// ---- Data types/Robot_udts/udt_GenericRobot_AnyFieldbus_OutputBytes_20220421.TcDUT
(*udt (user defined type) for all Fieldbus Based Robot Interfacing up to 64 Bytes
	Author(S): Brent Lekx-Toniolo of Sodecia GTAC;
	Version 1.0: November 2012
		- Initial Concept
	Version 20121204
		Changes from v1
			- Change to Naming Convention to include date as version
	Version 20220421
			- Changed starting point of Array fro 1 to 0 for TcHmi conventions, b.lekx-toniolo
*)
TYPE udt_GenericRobot_AnyFieldbus_OutputBytes_20220421 :
STRUCT
	Byte_: ARRAY [0..64] OF BYTE;
END_STRUCT
END_TYPE

// ---- Data types/Robot_udts/udt_GenericRobot_CycleTimes_20170304.TcDUT
(*udt (user defined type) for generic framework of cycle time counters for any robot
	Author(S): Brent Lekx-Toniolo of Sodecia GTAC;
	Version 20150622
		- Initila concept, BLT
	Version 20170304
		-added human, equip and total cycle time, JVD
*)
TYPE udt_GenericRobot_CycleTimes_20170304 :
STRUCT
	(*Cycle Times for Equipment Interf Zones*)
		Cycle_Time_OutEquip1: TIME;
		PrevCycle_Time_OutEquip1: TIME;
		Cycle_Time_OutEquip2: TIME;
		PrevCycle_Time_OutEquip2: TIME;
		Cycle_Time_OutEquip3: TIME;
		PrevCycle_Time_OutEquip3: TIME;
		Cycle_Time_OutEquip4: TIME;
		PrevCycle_Time_OutEquip4: TIME;
		Cycle_Time_OutEquip5: TIME;
		PrevCycle_Time_OutEquip5: TIME;
		Cycle_Time_OutEquip6: TIME;
		PrevCycle_Time_OutEquip6: TIME;
		Cycle_Time_OutEquip7: TIME;
		PrevCycle_Time_OutEquip7: TIME;
		Cycle_Time_OutEquip8: TIME;
		PrevCycle_Time_OutEquip8: TIME;

	(*Cycle Times for Human Interf Zones*)
		Cycle_Time_OutHuman1: TIME;
		PrevCycle_Time_OutHuman1: TIME;
		Cycle_Time_OutHuman2: TIME;
		PrevCycle_Time_OutHuman2: TIME;
		Cycle_Time_OutHuman3: TIME;
		PrevCycle_Time_OutHuman3: TIME;
		Cycle_Time_OutHuman4: TIME;
		PrevCycle_Time_OutHuman4: TIME;
		Cycle_Time_OutHuman5: TIME;
		PrevCycle_Time_OutHuman5: TIME;
		Cycle_Time_OutHuman6: TIME;
		PrevCycle_Time_OutHuman6: TIME;
		Cycle_Time_OutHuman7: TIME;
		PrevCycle_Time_OutHuman7: TIME;
		Cycle_Time_OutHuman8: TIME;
		PrevCycle_Time_OutHuman8: TIME;

		Cycle_Time_EquipTotal: TIME;
		Cycle_Time_HumanTotal: TIME;
		Cycle_Time_Total: TIME;

END_STRUCT
END_TYPE

// ---- Data types/Robot_udts/udt_Profibus_Motoman_Input.TcDUT
TYPE udt_Profibus_Motoman_Input :
	STRUCT
		Inputs:udt_ProfiNode_Status;
		(*Output Data From Robot*)
		SYS:UDINT;
		OG4: BYTE;
		OG5: BYTE;
		OG6: BYTE;
		OG7: BYTE;
		OG8: BYTE;
		OG9: BYTE;
		OG10: BYTE;
		OG11: BYTE;
		OG12: BYTE;
		OG13: BYTE;
		OG14: BYTE;
		OG15: BYTE;
		OG16: BYTE;
		OG17: BYTE;
		OG18: BYTE;
		OG19: BYTE;
		OG20: BYTE;
		OG21: BYTE;
		OG22: BYTE;
		OG23: BYTE;
		OG24: BYTE;
		OG25: BYTE;
		OG26: BYTE;
		OG27: BYTE;
		OG28: BYTE;
		OG29: BYTE;
		OG30: BYTE;
		OG31: BYTE;
		OG32: BYTE;
	END_STRUCT
END_TYPE

// ---- Data types/Robot_udts/udt_Profibus_Motoman_Input_20121204.TcDUT
(*udt (user defined type) for all Motoman Robot Controllers with HMS AnyBus Profibus Interface Card
	Author(S): Brent Lekx-Toniolo/Rob Remillard of Sodecia GTAC;
	Version 1.0: August 2010
		- Initial Concept
	Version 20121204
		Changes from v1
			- Increased Size to 32 Bytes
			- Change to Naming Convention to include date as version

	Last Edit: December 4th, 2012, blt
*)

TYPE udt_Profibus_Motoman_Input_20121204 :
	STRUCT
		Inputs:udt_ProfiNode_Status;
		(*Output Data From Robot, 32 Bytes total size*)
		SYS:UDINT;
		OG4: BYTE;
		OG5: BYTE;
		OG6: BYTE;
		OG7: BYTE;
		OG8: BYTE;
		OG9: BYTE;
		OG10: BYTE;
		OG11: BYTE;
		OG12: BYTE;
		OG13: BYTE;
		OG14: BYTE;
		OG15: BYTE;
		OG16: BYTE;
		OG17: BYTE;
		OG18: BYTE;
		OG19: BYTE;
		OG20: BYTE;
		OG21: BYTE;
		OG22: BYTE;
		OG23: BYTE;
		OG24: BYTE;
		OG25: BYTE;
		OG26: BYTE;
		OG27: BYTE;
		OG28: BYTE;
		OG29: BYTE;
		OG30: BYTE;
		OG31: BYTE;
		OG32: BYTE;
		OG33: BYTE;
	END_STRUCT
END_TYPE

// ---- Data types/Robot_udts/udt_Profibus_Motoman_Output.TcDUT
TYPE udt_Profibus_Motoman_Output :
	STRUCT
		(*Input Data To Robot*)
		SYS:UDINT;
		IG4:BYTE;
		IG5:BYTE;
		IG6:BYTE;
		IG7:BYTE;
		IG8:BYTE;
		IG9:BYTE;
		IG10:BYTE;
		IG11:BYTE;
		IG12:BYTE;
		IG13:BYTE;
		IG14:BYTE;
		IG15:BYTE;
		IG16:BYTE;
		IG17:BYTE;
		IG18:BYTE;
		IG19:BYTE;
		IG20:BYTE;
		IG21:BYTE;
		IG22:BYTE;
		IG23:BYTE;
		IG24:BYTE;
		IG25:BYTE;
		IG26:BYTE;
		IG27:BYTE;
		IG28:BYTE;
		IG29:BYTE;
		IG30:BYTE;
		IG31:BYTE;
		IG32:BYTE;
		END_STRUCT
END_TYPE

// ---- Data types/Robot_udts/udt_Profibus_Motoman_Output_20121204.TcDUT
(*udt (user defined type) for all Motoman Robot Controllers with HMS AnyBus Profibus Interface Card
	Author(S): Brent Lekx-Toniolo/Rob Remillard of Sodecia GTAC;
	Version 1.0: August 2010
		- Initial Concept
	Version 20121204
		Changes from v1
			- Increased Size to 32 Bytes
			- Change to Naming Convention to include date as version

	Last Edit: December 4th, 2012, blt
*)
TYPE udt_Profibus_Motoman_Output_20121204 :
	STRUCT
		(*Input Data To Robot, 32 Bytes total size*)
		SYS:UDINT;
		IG4:BYTE;
		IG5:BYTE;
		IG6:BYTE;
		IG7:BYTE;
		IG8:BYTE;
		IG9:BYTE;
		IG10:BYTE;
		IG11:BYTE;
		IG12:BYTE;
		IG13:BYTE;
		IG14:BYTE;
		IG15:BYTE;
		IG16:BYTE;
		IG17:BYTE;
		IG18:BYTE;
		IG19:BYTE;
		IG20:BYTE;
		IG21:BYTE;
		IG22:BYTE;
		IG23:BYTE;
		IG24:BYTE;
		IG25:BYTE;
		IG26:BYTE;
		IG27:BYTE;
		IG28:BYTE;
		IG29:BYTE;
		IG30:BYTE;
		IG31:BYTE;
		IG32:BYTE;
		IG33:BYTE;
		END_STRUCT
END_TYPE

// ---- Data types/Robot_udts/udt_SingleAxis_MoveData_20160908.TcDUT
(*udt (user defined type) to create data type for storing single Axis Movement Data Parameters:
	
	Author(S): Brent Lekx-Toniolo of Sodecia GTAC;

	Version 20150119
		- Initial Concept
	Version 20160908
		- Added Move_Type for vel vs pos type moves, b.lekx-toniolo


*)



TYPE udt_SingleAxis_MoveData_20160908 :
STRUCT
		Move_Type: UINT; 	(*Specify Move type during teaching*)
		Position: LREAL; 		(*Actual Stored Position Data*)
		Velocity: REAL; 		(*Target Velocity*)
		Accel: REAL; 			(*Target Acceleration Rate*)
		Decel: REAL;			(*Target Decceleration Rate*)
		End_Flag: BOOL;		(*Flag to Indicate Last Step In Program*)
END_STRUCT
END_TYPE

// ---- Data types/Robot_udts/udt_SingleAxis_Position_20150119.TcDUT
(*udt (user defined type) to create data type for storing single Axis Positional Data Parameters:
	
	Author(S): Brent Lekx-Toniolo of Sodecia GTAC;

	Version 20150119
		- Initial Concept

*)



TYPE udt_SingleAxis_Position_20150119 :
STRUCT
		Position: LREAL; 	(*Actual Stored Position Data*)
		Velocity: REAL; 	(*Target Velocity*)
		Accel: REAL; 		(*Target Acceleration Rate*)
		Decel: REAL;		(*Target Decceleration Rate*)
		End_Flag: BOOL;	(*Flag to Indicate Last Step In Program*)
END_STRUCT
END_TYPE

// ---- Data types/Schneider udts/udt_Schneider_VFD_20180808.TcDUT
(*udt (user defined type) for Schneider Electric VFD I/O Module
	Author(S): Justin Vandongen of Sodecia GTAC;

------------------------------------------------------------------------
	REVISION NOTES:

	Version 20180808
		- Initial Concept, j.vandongen
		- tested on ATV320 v1.11 ethercat module from schneider, j.vandongen

------------------------------------------------------------------------
*)

TYPE udt_Schneider_VFD_20180808 :
	STRUCT
	 	InfoData: udt_ECATSlave_Status;
	END_STRUCT
END_TYPE

// ---- Data types/Schneider udts/udt_Schneider_VFD_Image_20180808.TcDUT
(*udt (user defined type) for Schneider Electric VFD I/O Module
	Author(S): Justin Vandongen of Sodecia GTAC;

------------------------------------------------------------------------
	REVISION NOTES:

	Version 20180808
		- Initial Concept, j.vandongen
		- tested on ATV320 v1.11 ethercat module from schneider, j.vandongen
	Version 20250828
		- Added Cable breaks, r.jones
------------------------------------------------------------------------
*)

TYPE udt_Schneider_VFD_Image_20180808 :
	STRUCT
		
	VFD_State: udt_Schneider_VFD_20180808;
	Status_Word: UINT;
	Control_Word: UINT;
	Target_Velocity: INT;
	Move_TIME: TIME;
	ECAT_Cable_Breaks: UDINT;

	END_STRUCT
END_TYPE

// ---- Data types/Schneider udts/udt_Schneider_VFD_Inputs_20190123.TcDUT
(*udt (user defined type) for Schneider Electric VFD I/O Module
	Author(S): Justin Vandongen of Sodecia GTAC;

------------------------------------------------------------------------
	REVISION NOTES:

	Version 20180808
		- Initial Concept, j.vandongen
		- tested on ATV320 v1.11 ethercat module from schneider, j.vandongen
	Version 20190123
		- re-organized for more consistancy to generic device udts, b.lekx-toniolo

------------------------------------------------------------------------
*)

TYPE udt_Schneider_VFD_Inputs_20190123 :
	STRUCT
	InfoData: udt_ECATSlave_StatusEXT;

	Status_Word: UINT;
	Control_Effort: INT;
	Move_Time: TIME;

	END_STRUCT
END_TYPE

// ---- Data types/Schneider udts/udt_Schneider_VFD_Outputs_20190123.TcDUT
(*udt (user defined type) for Schneider Electric VFD I/O Module
	Author(S): Justin Vandongen of Sodecia GTAC;

------------------------------------------------------------------------
	REVISION NOTES:

	Version 20180808
		- Initial Concept, j.vandongen
		- tested on ATV320 v1.11 ethercat module from schneider, j.vandongen
	Version 20190123
		- re-organized for more consistancy to generic device udts, b.lekx-toniolo
------------------------------------------------------------------------
*)

TYPE udt_Schneider_VFD_Outputs_20190123 :
	STRUCT
	Control_Word: UINT;
	Target_Velocity: INT;
	END_STRUCT
END_TYPE

// ---- Data types/Servo Drive udts/AX5000 Diag/udt_AX5000Diag.TcDUT
(*Created by Beckhoff*)

TYPE udt_AX5000Diag :
STRUCT
	(* NC-Status *)
	nNCAxisID				: UDINT;
	bOperational				: BOOL;
	bC1DError				: BOOL;
	bWcStateError			: BOOL;
	bAxisError				: BOOL;
	iAxisErrorCode			: UDINT;

	(* Drive Diag *)
	strDriveType				: STRING(19);
	strMotorType				:STRING(31);
	wDriveStatus				: WORD;
	wClass1Diag				: WORD;
	stClass1Diag				: ST_AX5000_C1D;
	stDriveStatus				: ST_AX5000DriveStatus;
	stEcSlaveStateBits		: ST_EcSlaveStateBits;
	stEcSlaveState			: ST_EcSlaveState;
	bPreopToSafeOpError		: BOOL;
	bSafeOpToOpError		: BOOL;
	stCPxInvParamList			:ST_SoE_CPxInvParamList;
	iDiagNumber				: UDINT;
	stDiagNumberList			:ST_SoE_DiagNumList;
	strDiagMessage			: STRING(19);
	strDiagMessageFull		: STRING(60);
END_STRUCT
END_TYPE

// ---- Data types/Servo Drive udts/udt_AX5206_20160804.TcDUT
(*udt (user defined type) of Beckhoff AX5206 2 Axis Drive:
	auth. R.Remillard; 
	Oct 2014; version 1.0

	Version 20160804
		- Updated naming per convention, b.lekx-toniolo
		- Re-arranged variables for more consitent order with HW spec, b.lekx-toniolo
*)


TYPE udt_AX5206_20160804 :
STRUCT

	WcState:	BOOL;
	InfoData: udt_ECATSlave_StatusEXT;

END_STRUCT
END_TYPE

// ---- Data types/Servo Drive udts/udt_AX5805_20160804.TcDUT
(*udt (user defined type) of Beckhoff Type AX5805 Drive Safety Module:
	auth. R.Remillard; 
	October 2014; version 1.0

	Version 20160804
		- Updated naming per convention, b.lekx-toniolo
		- Re-arranged variables for more consitent order with HW spec, b.lekx-toniolo
	*)

TYPE udt_AX5805_20160804 :
STRUCT

	WcState:							BOOL;
 	InfoData: udt_ECATSlave_StatusEXT;

	FSOE_Command: 					USINT;
	Axis1_STO:						BOOL;
	Axis1_SSM1:						BOOL;
	Axis1_SSM2:						BOOL;
	Axis1_SOS1:						BOOL;
	Axis1_SSR1:						BOOL;
	Axis1_SDIp:						BOOL;
	Axis1_SDIn:						BOOL;
	Axis1_Error_Ack:					BOOL;
	FSOE_Slave_CRC_0:				UINT;
	Axis2_STO:						BOOL;
	Axis2_SSM1:						BOOL;
	Axis2_SSM2:						BOOL;
	Axis2_SOS1:						BOOL;
	Axis2_SSR1:						BOOL;
	Axis2_SDIp:						BOOL;
	Axis2_SDIn:						BOOL;
	Axis2_Error_Ack:					BOOL;
	FSOE_Slave_CRC_1:				UINT;
	FSOE_ConnID:					UINT;

	AMSAddress:						udt_AdsAddr_AX5805;

END_STRUCT
END_TYPE

// ---- Data types/Servo Drive udts/udt_AX5805_DiagData.TcDUT
TYPE udt_AX5805_DiagData :
STRUCT
	InternalDataA1:		UINT;	(*STO Reason Code Axis 1*)
	InternalDataA2:		UINT;	(*STO Reason Code Axis 2*)
	DiagDataA1:			UINT;	(*Ax5805 Setup Diagnositcs Axis 1*)
	DiagDataA2:			UINT;	(*AX5805 Setup Diagnostics Axis 2*)
	bError:				BOOL;
END_STRUCT
END_TYPE

// ---- Data types/Servo Drive udts/udt_EL7211_20150115.TcDUT
(*udt (user defined type) of Beckhoff - EL7211 series servo terminals:
	
	Author(S): Brent Lekx-Toniolo of Sodecia GTAC;

	Version 20150115
		- Initial Concept

*)


TYPE udt_EL7211_20150115 :
	STRUCT
		InfoData: udt_ECATSlave_Status;
	END_STRUCT
END_TYPE

// ---- Data types/SIC/udt_SIC_Profi_Input_20200727.TcDUT
TYPE udt_SIC_Profi_Input_20200727 :
STRUCT

			(*Status Of Profibus Slave*)
		Inputs:udt_ProfiNode_Status;
		(*Input Bytes*)
		Input0_0: ARRAY [0..15] OF USINT;
		Input0_1: ARRAY [0..15] OF USINT;
		Input0_2: ARRAY [0..15] OF USINT;
		Input0_3: ARRAY [0..15] OF USINT;
		Input0_4: ARRAY [0..15] OF USINT;
		Input0_5: ARRAY [0..15] OF USINT;
		Input0_6: ARRAY [0..15] OF USINT;
		Input0_7: ARRAY [0..15] OF USINT;
		Input0_8: ARRAY [0..15] OF USINT;
		Input0_9: ARRAY [0..15] OF USINT;
		Input0_10: ARRAY [0..15] OF USINT;
		Input0_11: ARRAY [0..15] OF USINT;
		Input0_12: ARRAY [0..15] OF USINT;
		Input0_13: ARRAY [0..15] OF USINT;
		Input0_14: ARRAY [0..15] OF USINT;
		Input0_15: ARRAY [0..15] OF USINT;

END_STRUCT
END_TYPE

// ---- Data types/SIC/udt_SIC_Profi_Output_20200727.TcDUT
TYPE udt_SIC_Profi_Output_20200727 :
STRUCT
	

		(*Input Bytes*)
		Output1_0: ARRAY [0..15] OF USINT;
		Output1_1: ARRAY [0..15] OF USINT;
		Output1_2: ARRAY [0..15] OF USINT;
		Output1_3: ARRAY [0..15] OF USINT;
		Output1_4: ARRAY [0..15] OF USINT;
		Output1_5: ARRAY [0..15] OF USINT;
		Output1_6: ARRAY [0..15] OF USINT;
		Output1_7: ARRAY [0..15] OF USINT;
		Output1_8: ARRAY [0..15] OF USINT;
		Output1_9: ARRAY [0..15] OF USINT;
		Output1_10: ARRAY [0..15] OF USINT;
		Output1_11: ARRAY [0..15] OF USINT;
		Output1_12: ARRAY [0..15] OF USINT;
		Output1_13: ARRAY [0..15] OF USINT;
		Output1_14: ARRAY [0..15] OF USINT;
		Output1_15: ARRAY [0..15] OF USINT;
		
END_STRUCT
END_TYPE

// ---- Data types/SmartRay/udt_PLC_Out_To_SmartRay_IN_20260119.TcDUT
(*udt of SmartRay profinet based
    PLC > Smart Ray 
  auth . Sodecia GTAC;
  Jan 2026: Version 1.0*)
TYPE udt_PLC_Out_To_SmartRay_IN_20260119 :
	
STRUCT
	(*Byte 0*)
	Byte_0 : BYTE;
	//PartType_In : BYTE;
	
	(*Byte 2-21*)
	Byte_2_21 : ARRAY[0..19] OF BYTE;
    //PartID_In : ARRAY[0..19] OF BYTE;
	
	(*Byte 24-43*)
	Byte_24_43 : ARRAY[0..19] OF BYTE;
	//PartIDVisu1_In : ARRAY[0..19] OF BYTE;
		
	(*Byte 44*)
	Byte_44 : BYTE;
	//Visu_NextPage_In : BOOL; (*Bit 4*)
	//Visu_NextWeld_In : BOOL; (*Bit 5*)
	//Visu_PreviousWeld_In : BOOL; (*Bit 6*)
	
	(*Byte 45*)
	Byte_45 : BYTE;
	//Visu_WorkerButton_In : BYTE; 
	
	(*Byte 48-67*)
	Byte_48_67 : ARRAY[0..19] OF BYTE;
	//PartIDVisu2_In : ARRAY[0..19] OF BYTE;
	
	(*Byte 68*)
	Byte_68 : BYTE;
	//Visu_NextPage2_In : BOOL; (*Bit 4*)
	//Visu_NextWeld2_In : BOOL; (*Bit 5*)
	//Visu_PreviousWeld2_In : BOOL; (*Bit 6*)

	(*Byte 69*)
	Byte_69 : BYTE;
	//Visu_WorkerButton2_In : BYTE;

END_STRUCT
END_TYPE

// ---- Data types/SmartRay/udt_Robot_Out_To_SmartRay_IN_20260119.TcDUT
TYPE udt_Robot_Out_To_SmartRay_IN_20260119 :
	// udt : Robot > Smart Ray
STRUCT
	(*Byte 0*)
	Reset_In : BOOL; (*Bit 0*)
	Alive_In : BOOL; (*Bit 1*)
	AutomaticMode_In : BOOL; (*Bit 2*)
 	SetupMode_In : BOOL; (*Bit 3*)
	
	(*Byte 1*)
	LaserOn_In : BOOL; (*Bit 1*)
	LaserOn2_In : BOOL; (*Bit 2*)
	SensortestOn_In : BOOL; (*Bit 3*)
	
	(*Byte 2*)
	InspectionCompleted_In : BOOL; (*Bit 2*)
	ToolfinderOn_In : BOOL; (*Bit 4*)

	(*Byte 3*)
	RobotSelection_In : BYTE;
	
	(*Byte 4-5*)
	JobID_In : UINT;
	
	(*Byte 6-7*)
	TrackSpeed_In : UINT;
	
END_STRUCT
END_TYPE

// ---- Data types/SmartRay/udt_SmartRay_Out_To_PLC_IN_20260119.TcDUT
(*udt of SmartRay profinet based
   Smart Ray > PLC 
  auth . Sodecia GTAC;
  Jan 2026: Version 1.0*)
TYPE udt_SmartRay_Out_To_PLC_IN_20260119 :
STRUCT
	(*Byte 0*)
	Byte_0 : BYTE;
	//PartType_Out : BYTE;
	
	(*Byte 2-21*)
	Byte_2_21 : ARRAY[0..19] OF BYTE;
	//PartID_Out : ARRAY[0..19] OF BYTE;
	
	(*Byte 22*)
	Byte_22 : BYTE;
	//QualityOK_Out_2 : BOOL; (*Bit 0*)
	//QualityNOK_Out_2 : BOOL; (*Bit 1*)
	//ResultValid_Out_2 : BOOL; (*Bit 2*)
	//LastTelegramSent_Out : BOOL; (*Bit 7*)
	
	(*Byte 24-43*)
	Byte_24_43 : ARRAY[0..19] OF BYTE;
	//PartIDVisu1_Out : ARRAY[0..19] OF BYTE;
	
	(*Byte 44*)
	Byte_44 : BYTE;
	(*WorkerResultOK_Out : BOOL; (*Bit 0*)
	WorkerResultNOK_Out : BOOL; (*Bit 1*)
	ReworkOK_Out : BOOL; (*Bit 2*)
	ReworkDone_Out : BOOL; (*Bit 3*)
	Visu_NextPage_Out : BOOL; (*Bit 4*)
	Visu_NextWeld_Out : BOOL; (*Bit 5*)
	Visu_PreviousWeld_Out : BOOL; (*Bit 6*)*)
	
	(*Byte 45*)
	Byte_45 : BYTE;
	//Visu_WorkerButon_Out :BYTE; 
	
	(*Byte 48-67*)
	Byte_48_67 : ARRAY[0..19] OF BYTE;
	//PartIDVisu2_Out : ARRAY[0..19] OF BYTE;
	
	(*Byte 68*)
	Byte_68 : BYTE;
	(*WorkerResultOK2_Out : BOOL; (*Bit 0*)
	WorkerResultNOK2_Out : BOOL; (*Bit 1*)
	ReworkOK2_Out : BOOL; (*Bit 2*)
	ReworkDone2_Out : BOOL; (*Bit 3*)
	Visu_NextPage2_Out : BOOL; (*Bit 4*)
	Visu_NextWeld2_Out : BOOL; (*Bit 5*)
	Visu_PreviousWeld2_Out : BOOL; (*Bit 6*)*)
	
	(*Byte 69*)
	Byte_69 : BYTE;
	//Vis_WorkerButton2_Out : BYTE;
	
	(*Byte 80-179*)
	Byte_80_179 : ARRAY[0..99] OF BYTE;
	//WeldResult_Out : ARRAY[0..99] OF BYTE;

END_STRUCT
END_TYPE

// ---- Data types/SmartRay/udt_SmartRay_Out_To_Robot_IN_20260119.TcDUT
(*udt of SmartRay profinet based
   Smart Ray > Robot 
  auth . Sodecia GTAC;
  Jan 2026: Version 1.0*)
TYPE udt_SmartRay_Out_To_Robot_IN_20260119 :	
STRUCT
	(*Status*)
	(*Byte 0*)
	SystemReady_Out : BOOL; (*Bit 0*)
	Alive_Out : BOOL; (*Bit 1*)
    FailureSystem_Out : BOOL; (*Bit 4*)
	FailureGlobal_Out : BOOL; (*Bit 5*)
	
	(*Byte 1*)
	SensorReady_Out : BOOL; (*Bit 0*)
	LaserOn_Out : BOOL; (*Bit 1*)
	LaserOn2_Out : BOOL; (*Bit 2*)
	SensortestOK_Out : BOOL; (*Bit 4*)
	SensortestNOK_Out : BOOL; (*Bit 5*)
	
	(*Byte 2*)
	QualityOK_Out : BOOL; (*Bit 0*)
	QualityNOK_Out : BOOL; (*Bit 1*)
	InspectionCompleted_Out : BOOL;(*Bit 2*)
	ResultValid_Out : BOOL; (*Bit 3*)
	ToolfinderValid_Out : BOOL; (*Bit 4*)
	ReferenceTrackSpeedActive_Out : BOOL; (*Bit 5*)
	
	(*Byte 3*)
	RobotSelection_Out : BYTE;
	
	(*Byte 4-5*)
	JobID_Out : UINT;
	
	(*Byte 6*)
	ErrorCode_Out : BYTE;
	
	(*Byte 7*)
	ToolfinderErrorCode_Out : BYTE;
	
	(*Byte 8-9*)
	Toolfinder_X : INT ;
	
	(*Byte 10-11*)
	Toolfinder_Y : INT;
	
	(*Byte 12-13*)
	Toolfinder_Z : INT;
	
	(*Byte 14-15*)
	Toolfinder_Q1_A_W :INT;
	
	(*Byte 16-17*)
	Toolfinder_Q2_B_P : INT;
	
	(*Byte 18-19*)
	Toolfinder_Q3_C_R : INT;
	
	(*Byte 20-21*)
	Toolfinder_Q4 : INT;
	
END_STRUCT
END_TYPE

// ---- Data types/SmartRay/UI udt/udt_SRxx_DiscreteImage.TcDUT
TYPE udt_SRxx_DiscreteImage :
STRUCT
	(*Smart Ray*)
	SR_Error : BOOL;
	SR_Comm_Error : BOOL;
	SR_PLC_FB_Error : BOOL;
	SR_Smart_Ray_OK : BOOL;
	SR_Smart_Ray_NOK : BOOL;
	
	Profinode_status : udt_ProfiNet_Status;

END_STRUCT
END_TYPE

// ---- Data types/SmartRay/UI udt/udt_SRxx_Input_Image.TcDUT
TYPE udt_SRxx_Input_Image :
STRUCT
	Retry : BOOL;
	Bypass :BOOL;
END_STRUCT
END_TYPE

// ---- Data types/SmartRay/UI udt/udt_SRxx_ToUI_20260122.TcDUT
TYPE udt_SRxx_ToUI_20260122 :
STRUCT
	DiscreteImage : udt_SRxx_DiscreteImage;
END_STRUCT
END_TYPE

// ---- Data types/SMC udts/udt_SMC_EX260_Stat.TcDUT
(*udt (user defined type) for SMC EX260 Serial Interface Valve Bank System EtherCAT Slave:
	auth. Brent Lekx-Toniolo of Toniolo Research & Development Inc.; 
	July 2010; version 1.0*)


TYPE udt_SMC_EX260_Stat :
STRUCT
	InfoData: udt_ECATSlave_Status;
END_STRUCT
END_TYPE

// ---- Data types/SMC udts/udt_SMC_EX260_ValveBank.TcDUT
(*udt (user defined type) for SMC EX260 Serial Interface Valve Bank System EtherCAT Slave:
	auth. Brent Lekx-Toniolo of Toniolo Research & Development Inc.; 
	August 2010; version 1.0*)


TYPE udt_SMC_EX260_ValveBank :
STRUCT
	Q: DINT;
END_STRUCT
END_TYPE

// ---- Data types/Trumpf udts/udt_EtherCat_Trumpf_InputWords_20171002.TcDUT

(*udt (user defined type) for all EtherCAT Based Trumpf Laser Interfacing on EL6692, up to 64 Bytes
	Author(S): Justin Vandongen of Sodecia GTAC;

------------------------------------------------------------------------
	REVISION NOTES:

	Version 20171002
		- Initial Concept, j.vandongen

------------------------------------------------------------------------
*)



TYPE udt_EtherCat_Trumpf_InputWords_20171002 :
STRUCT
	Laser_Out: ARRAY [0..9] OF WORD;
END_STRUCT
END_TYPE

// ---- Data types/Trumpf udts/udt_EtherCat_Trumpf_OutputWords_20171002.TcDUT

(*udt (user defined type) for all EtherCAT Based Trumpf Laser Interfacing on EL6692, up to 64 Bytes
	Author(S): Justin Vandongen of Sodecia GTAC;

------------------------------------------------------------------------
	REVISION NOTES:

	Version 20171002
		- Initial Concept, j.vandongen

------------------------------------------------------------------------
*)



TYPE udt_EtherCat_Trumpf_OutputWords_20171002 :
STRUCT
	Laser_In: ARRAY [0..9] OF WORD;
END_STRUCT
END_TYPE

// ---- Data types/Trumpf udts/udt_TrumpfImage_20171017.TcDUT

(*udt (user defined type) for all EtherCAT Based Trumpf Laser Discrete I/O Module
	Author(S): Justin Vandongen of Sodecia GTAC;

------------------------------------------------------------------------
	REVISION NOTES:

	Version 20171017
		- Initial Concept, j.vandongen

------------------------------------------------------------------------
*)


TYPE udt_TrumpfImage_20171017 :
STRUCT

		LSRT01: udt_EL6692_20121204;	(*EtherCAT bridge for Laser controller*)

		Program_REQ: UDINT;
		Program_ACK: UDINT;

		Light_Path_REQ: UDINT;
		Light_Path_ACK: UDINT;

		Laser_No_REQ: UDINT;
		Laser_No_ACK: UDINT;

		Laser_Power: UDINT;
		Laser_Power_Prev: UDINT;
		Energy: UDINT;
		Energy_Prev: UDINT;

		Weld_Complete: BOOL;
		Faulted: BOOL;


END_STRUCT
END_TYPE

// ---- Data types/UI udts/GTAC Component IO UI udts/udt_IVxx_ToUI_20250808.TcDUT
(*udt (user defined type) for interfacing to UI (User Interface)
this udt represents data that is passed from PLC to EACH UI

	Author(S): R.jones of Sodecia GTAC;
	- Initial Concept
	Version 20250723

*)

TYPE udt_IVxx_ToUI_20250808 :
	STRUCT

	(*Input and Output Data Images*)
	Discrete_Image: udt_IV2_DiscreteImage;
	(*EtherCAT Cable Break Flags*)
	ECAT_Cable_Breaks: UDINT;

	END_STRUCT
END_TYPE

// ---- Data types/UI udts/GTAC Component IO UI udts/udt_LSRxx_ToUI_20220224.TcDUT
(*udt (user defined type) for interfacing to UI (User Interface)
this udt represents data that is passed from PLC to EACH UI

	Author(S): Justin Vandongen of Sodecia GTAC;
	Version 20171011
		- Initial Concept
	Version 20220224
	- Overhaul during TcUI Migration project, b.lekx-toniolo / c.drees
*)

TYPE udt_LSRxx_ToUI_20220224:
	STRUCT

	(*Input and Output Data Images*)
	In_Image: udt_EtherCat_Trumpf_InputWords_20171002;
	Out_Image: udt_EtherCat_Trumpf_OutputWords_20171002;
	Discrete_Image: udt_TrumpfImage_20171017;

	(*EtherCAT Cable Break Flags*)
	ECAT_Cable_Breaks: UDINT;

	UI_FaultPrompts: UDINT;

	END_STRUCT
END_TYPE

// ---- Data types/UI udts/GTAC Component IO UI udts/udt_ESWxx_ToUI_20220224.TcDUT
(*udt (user defined type) for interfacing to UI (User Interface)
this udt represents data that is passed from PLC to EACH UI

	Author(S): Brent Lekx-Toniolo of Sodecia GTAC;
	Version 20150814
		- Initial Concept
	Version 20220224
	- Overhaul during TcUI Migration project, b.lekx-toniolo / c.drees

*)

TYPE udt_ESWxx_ToUI_20220224 :
	STRUCT

	(*Input and Output Data Images*)
	Discrete_Image: udt_ESWxx_Image_20150814;
	(*EtherCAT Cable Break Flags*)
	ECAT_Cable_Breaks: UDINT;

	END_STRUCT
END_TYPE

// ---- Data types/UI udts/GTAC Component IO UI udts/udt_ICxx_ToUI_20220224.TcDUT
(*udt (user defined type) for interfacing to UI (User Interface)
this udt represents data that is passed from PLC to EACH UI

	Author(S): Brent Lekx-Toniolo of Sodecia GTAC;
	Version 20141020
		- Initial Concept
	Version 20220224
	- Overhaul during TcUI Migration project, b.lekx-toniolo / c.drees

*)

TYPE udt_ICxx_ToUI_20220224 :
	STRUCT

	(*Input and Output Data Images*)
	Discrete_Image: udt_ICxx_Image;
	(*EtherCAT Cable Break Flags*)
	ECAT_Cable_Breaks: UDINT;

	END_STRUCT
END_TYPE

// ---- Data types/UI udts/GTAC Component IO UI udts/udt_MDxx_ToUI_20251008.TcDUT
(*udt (user defined type) for interfacing to UI (User Interface)
this udt represents data that is passed from PLC to EACH UI

	Author(S): Brent Lekx-Toniolo of Sodecia GTAC;
	Version 20150814
		- Initial Concept
	Version 20240926
	- Overhaul during TcUI Migration project, b.lekx-toniolo
	Version 20251008
	- MDxx instance update, b.lekx-toniolo
*)

TYPE udt_MDxx_ToUI_20251008 :
	STRUCT

	(*Input and Output Data Images*)
	Discrete_Image: udt_MDxx_Image_20251008;
	(*EtherCAT Cable Break Flags*)
	ECAT_Cable_Breaks: UDINT;

	END_STRUCT
END_TYPE

// ---- Data types/UI udts/GTAC Component IO UI udts/udt_NWxx_ToUI_20220224.TcDUT
(*udt (user defined type) for interfacing to UI (User Interface)
this udt represents data that is passed from PLC to EACH UI

	Author(S): Brent Lekx-Toniolo of Sodecia GTAC;
	Version 20141020
		- Initial Concept
	Version 20220224
	- Overhaul during TcUI Migration project, b.lekx-toniolo / c.drees

*)

TYPE udt_NWxx_ToUI_20220224 :
	STRUCT

	(*Input and Output Data Images*)
	Discrete_Image: udt_NWx_Image;
	(*EtherCAT Cable Break Flags*)
	ECAT_Cable_Breaks: UDINT;

	END_STRUCT
END_TYPE

// ---- Data types/UI udts/GTAC Component IO UI udts/udt_ISxx_ToUI_20241121.TcDUT
(*udt (user defined type) for interfacing to UI (User Interface)
this udt represents data that is passed from PLC to EACH UI

	Author(S): Brent Lekx-Toniolo of Sodecia GTAC;
	Version 20150813
		- Initial Concept
	Version 20220224
	- Overhaul during TcUI Migration project, b.lekx-toniolo / c.drees
	Version 20241121
		-PD to IS rename, as per GH SSCC610 repo Issue#162, b.lekx-toniolo

*)

TYPE udt_ISxx_ToUI_20241121 :
	STRUCT

	(*Input and Output Data Images*)
	Discrete_Image: udt_ISxx_Image_20241121;
	(*EtherCAT Cable Break Flags*)
	ECAT_Cable_Breaks: UDINT;
	END_STRUCT
END_TYPE

// ---- Data types/UI udts/GTAC Component IO UI udts/udt_ProdReportxx_ToUI_20220224.TcDUT
(*udt (user defined type) for interfacing to UI (User Interface)
this udt represents data that is passed from PLC to EACH UI

	Author(S): Brent Lekx-Toniolo of Sodecia GTAC;
	Version 20141021
		- Initial Concept
	Version 20160229
		- Updated udt instances, b.lekx-toniolo
	Version 20191125
		- Updated udt instances, b.lekx-toniolo
	Version 20220224
	- Overhaul during TcUI Migration project, b.lekx-toniolo / c.drees

*)

TYPE udt_ProdReportxx_ToUI_20220224 :
	STRUCT
	Curr_Prod_Report: udt_Generic_Production_20221007;
	Days_Prod_Report: udt_Generic_Production_20221007;
	Aft_Prod_Report: udt_Generic_Production_20221007;
	Mid_Prod_Report: udt_Generic_Production_20221007;

	END_STRUCT
END_TYPE

// ---- Data types/UI udts/GTAC Component IO UI udts/udt_Rxx_ToUI_20220224.TcDUT
(*udt (user defined type) for interfacing to UI (User Interface)
this udt represents data that is passed from PLC to EACH UI

	Author(S): Rob Remillard/Brent Lekx-Toniolo of Sodecia GTAC;
	Version 20121204
		- Initial Concept
		- For use with Generic Robot Image + ASSCV4.6, None SafeOP Discrete Image
	Version 20141020
		- Modified Name During Addition of more devices, b.lekx-toniolo
	Version 20150622
		- Added variables for passing of Interf Cycle Times, b.lekx-toniolo
	Version 20151028
		- Added discrete image type FSOE for V5.00 machine changes, b.lekx-toniolo
		- Added discrete image area for water stands, b.lekx-toniolo
	Version 20170531
		- Fronius Updates, b.lekx-toniolo
		- EOAT Instance Update, b.lekx-toniolo
	Version 20180418
		-EOAT instance removed, j.vandongen
	Version 20220224
	- Overhaul during TcUI Migration project, b.lekx-toniolo / c.drees

*)

TYPE udt_Rxx_ToUI_20220224 :
	STRUCT
	Robot_Type: UINT;
	(*General Data*)
	Status: UINT;
	Axis_Data: ARRAY [0..8] OF REAL;
 
	(*Input and Output Data Images*)
	In_Image: udt_GenericRobot_AnyFieldbus_InputBytes_20220421;
	Out_Image: udt_GenericRobot_AnyFieldbus_OutputBytes_20220421;
	Discrete_ImageFSOE: udt_RobotDiscreteNode_ImageFSOE_20151028;
	Discrete_ImageSSCCV46: udt_RobotDiscreteNode_ImageSSCCv46_20121204;
	Discrete_ImageSSCCV46wSAFEOP: udt_RobotDiscreteNode_ImageSSCCv46wSAFEOP_20131903;


	(*Option Configuration Inputs*)
	Options: udt_Generic_Robot_Options_20170531;
		(*Optional Equipment related to Robot*)
		WS_Discrete_Image: ARRAY [0..2] OF udt_WaterStand_Image_20220131;
		ATI_Discrete_Image: udt_ATIxx_Image_20151104;
		Reamer_Discrete_Image: udt_Reamerxx_Image_20180405;
		(*Robot Fronius Status Visualization*)
		Fronius_Status: udt_Fronius_Status_20170531;

	(*EtherCAT Cable Break Flags*)
	ECAT_Cable_Breaks: UDINT;
	(*Cycle Times*)
	CT: udt_GenericRobot_CycleTimes_20170304;
	(*Ped IO to be shown*)
	Ped_IO_ToShow: ARRAY [0..3] OF UINT;

	END_STRUCT
END_TYPE

// ---- Data types/UI udts/GTAC Component IO UI udts/udt_SDxx_ToUI_20220224.TcDUT
(*udt (user defined type) for interfacing to UI (User Interface)
this udt represents data that is passed from PLC to EACH UI

	Author(S): Rob Remillard/Brent Lekx-Toniolo of Sodecia GTAC;
	Version 2015 (Named udt_HMI_Input): August 2010
		- Initial Concept
	Version 20160804
		- Renamed to "...UI specific_SD...." for convention, b.lekx-toniolo
		- Added Data area for Positioning UI, b.lekx-toniolo
		- Updated instance of drive image as per it's naming update, b.lekx-toniolo
	Version 20220224
	- Overhaul during TcUI Migration project, b.lekx-toniolo / c.drees

*)

TYPE udt_SDxx_ToUI_20220224 :
	STRUCT

		(*Input and Output Data Images*)
		Discrete_Image:	udt_Drive_Image_20190816;
		(*EtherCAT Cable Break Flags*)
		ECAT_Cable_Breaks: UDINT;
		(*Confirm Axis Local Control Request*)
		AxisLocalControl_IC_ACKS: ARRAY[0..2] OF UINT;

	END_STRUCT
END_TYPE

// ---- Data types/UI udts/GTAC Component IO UI udts/udt_SLxx_ToUI_20220224.TcDUT
(*udt (user defined type) for interfacing to UI (User Interface)
this udt represents data that is passed from PLC to EACH UI

	Author(S): Brent Lekx-Toniolo of Sodecia GTAC;
	Version 20141020
		- Initial Concept
	Version 20220224
	- Overhaul during TcUI Migration project, b.lekx-toniolo / c.drees

*)

TYPE udt_SLxx_ToUI_20220224 :
	STRUCT

	(*Input and Output Data Images*)
	In_Image: udt_Graco_Input;
	Out_Image: udt_Graco_Outputs;
	(*Image for Profibus Master (Internal or External to Dispensing unit)*)
	Txx_ProfiMaster AT %I*: udt_EL6731;
	(*EtherCAT Cable Break Flags*)
	ECAT_Cable_Breaks: UDINT;


	END_STRUCT
END_TYPE

// ---- Data types/UI udts/GTAC Component IO UI udts/udt_SSxx_ToUI_20250704.TcDUT
(*udt (user defined type) for interfacing to UI (User Interface)
this udt represents data that is passed from PLC to EACH UI

	Author(S): Brent Lekx-Toniolo of Sodecia GTAC;
	Version 20150814
		- Initial Concept
	Version 20220224
	- Overhaul during TcUI Migration project, b.lekx-toniolo / c.drees

*)

TYPE udt_SSxx_ToUI_20250704 :
	STRUCT

	(*Input and Output Data Images*)
	Discrete_Image: udt_SSxx_Image_20250704;
	(*EtherCAT Cable Break Flags*)
	ECAT_Cable_Breaks: UDINT;

	END_STRUCT
END_TYPE

// ---- Data types/UI udts/GTAC Component IO UI udts/udt_STxx_ToUI_20220224.TcDUT
(*udt (user defined type) for interfacing to UI (User Interface)
this udt represents data that is passed from PLC to EACH UI

	Author(S): Brent Lekx-Toniolo of Sodecia GTAC;
	Version 20141020
		- Initial Concept
	Version 20200212
		- Updated Instances for Nelson to Emhart changes, b.lekx-toniolo
	Version 20220224
	- Overhaul during TcUI Migration project, b.lekx-toniolo / c.drees

*)

TYPE udt_STxx_ToUI_20220224 :
	STRUCT

	(*Input and Output Data Images*)
	In_Image: udt_Emhart_TE1500_Input;
	Out_Image: udt_Emhart_TE1500_Output;
	Discrete_Image: udt_STxx_DiscreteNode_20200212;
	(*EtherCAT Cable Break Flags*)
	ECAT_Cable_Breaks: UDINT;


	END_STRUCT
END_TYPE

// ---- Data types/UI udts/GTAC Component IO UI udts/udt_SDxx_FromUI_20220224.TcDUT
(*udt (user defined type) for interfacing to UI (User Interface)
this udt represents data that is passed from EACH UI to PLC

	Author(S): Brent Lekx-Toniolo of Sodecia GTAC;
	Version 20160811
		- Original Concept, b.lekx-toniolo
	Version 20220224
	- Overhaul during TcUI Migration project, b.lekx-toniolo / c.drees

*)
TYPE udt_SDxx_FromUI_20220224 :
STRUCT
		AxisLocalControl_IC_REQS: ARRAY[0..2] OF UINT;
		Mode_Select: ARRAY[0..2] OF INT;
		Error_Reset: ARRAY[0..2] OF BOOL;
		Program_Reset: ARRAY[0..2] OF BOOL;

		PlayBack_Speed_Percentage: ARRAY[0..2] OF REAL;
		Explicit_Step_REQ: ARRAY[0..2] OF UINT;
		Start_Explicit_StepCall: ARRAY[0..2] OF BOOL;
		Start_PlayBack: ARRAY[0..2] OF BOOL;
		Stop_PlayBack: ARRAY[0..2] OF BOOL;
		PlayBack_StepPermit: ARRAY[0..2] OF BOOL;


		Teach_Params: ARRAY[0..2] OF udt_SingleAxis_MoveData_20160908; (*Struct of Teach paramaeters*)
		Teach_Servo_HomePos: ARRAY[0..2] OF BOOL;
		Teach_JogFast_Plus: ARRAY[0..2] OF BOOL;
		Teach_JogFast_Minus: ARRAY[0..2] OF BOOL;
		Teach_JogSlow_Plus: ARRAY[0..2] OF BOOL;
		Teach_JogSlow_Minus: ARRAY[0..2] OF BOOL;
		Teach_Inch_Plus: ARRAY[0..2] OF BOOL;
		Teach_Inch_Minus: ARRAY[0..2] OF BOOL;
		Teach_MicroInch_Enable: ARRAY[0..2] OF BOOL;
		Teach_Record_CurrentPos: ARRAY[0..2] OF BOOL;
		Teach_ParamsOverwrite_Flag: ARRAY[0..2] OF BOOL;

END_STRUCT
END_TYPE

// ---- Data types/UI udts/GTAC Component IO UI udts/udt_VFDxx_ToUI_20250723.TcDUT
(*udt (user defined type) for interfacing to UI (User Interface)
this udt represents data that is passed from PLC to EACH UI

	Author(S): Rich Jones;
	Version 20250723
	- Initial Concept
	
*)

TYPE udt_VFDxx_ToUI_20250723 :
	STRUCT

	(*Input and Output Data Images*)
	Discrete_Image: udt_Schneider_VFD_Image_20180808;

	END_STRUCT
END_TYPE

// ---- Data types/UI udts/udt_UIcommon_InputPers_20250612.TcDUT
(*udt (user defined type) for interfacing to UI (User Interface)
this udt represents PERSISTENT data that is passed from ALL UIs to PLC

	Version 20191127
		- Cleaned up various, added structure and added production config variables, b.lekx-toniolo
	Version 20250612
		- Added in Nut Weld LVDT Config area to help reduce ground up work on nut weld applications, b.lekx-toniolo
*)

TYPE udt_UIcommon_InputPers_20250612 :
	STRUCT
(*Standard Persistent Inputs from UI*)
	(*Production Configuration*)
	ProdConfig_Common: udt_Generic_ShiftCommonConfig_20220420;
	ProdConfig_Day: udt_Generic_ShiftConfigUDINT_20160531;
	ProdConfig_Aft: udt_Generic_ShiftConfigUDINT_20160531;
	ProdConfig_Mid: udt_Generic_ShiftConfigUDINT_20160531;

(*Nut Weld based LVDT Configuration*)
	Config_NutWeld_LVDT: ARRAY [0..5] OF udt_Generic_NutWeldLVDTConfig_20250612;
	
(*General QA Configuration Items*)
	Config_Vision_Fail_Limits: ARRAY[0..16] OF  UINT;
	Config_NOK_BinCount_Limits: ARRAY[0..16] OF UINT;
	Config_NOK_Consecutive_Limits: ARRAY[0..16] OF UINT;
	
	
(*Add Non- Standard Persistent Inputs from UI here*)


	END_STRUCT
END_TYPE

// ---- Data types/UI udts/udt_UIcommon_Input_20250616.TcDUT
(*udt (user defined type) for interfacing to UI (User Interface)
this udt represents data that is passed from ALL UIs to PLC

	Author(S): Rob Remillard/Brent Lekx-Toniolo of Sodecia GTAC;
	Version 1.0 (Named udt_HMI_Input): August 2010
		- Initial Concept
	Version 20141014
		- Increase for 30 Robot framework + Fix Renaming, b.lekx-toniolo
	Version 20150519
		- Added Report_Trigger_Reqs, b.lekx-toniolo
		- Added Rxx_ToolChange_Reqs, b.lekx-toniolo
	Version 20161129
		-Custom Setup for SIC marking, RRemillard
	Version 20161206
		-added Sealer bits, J.vandongen
	Version 20170626
		- added local dry cycle enables, b.lekx-toniolo / c.drees (edge automation)
	Version 20170801
		-added bit to control monitoring spaces from plc, RRemillard
	Version 20170804
		-added cycle hold, j.vandongen
	Version 20200611
		- added Rxx_Dress_Req, j.vandongen
	Version 20220224
		- overhaul during TcUI migration project, b.lekx-toniolo / c.drees
	Version 20240620
		- added rxx_tracctcp_req,  w. griffiths / b.lekx-toniolo 
	Version 20250616
		- Added in Nut Weld Based LVDT Input Image, b.lekx-toniolo	

*)

TYPE udt_UIcommon_Input_20250616 :
	STRUCT
(*Standard Inputs from UI*)
	(*Common to Cell*)
	StartRobots: BOOL;
	StopRobots: BOOL;
	Cycle_Hold: BOOL;
	RelaseSGK1: BOOL;
	RelaseSGK2: BOOL;
	LockSGK1: BOOL;
	LockSGK2: BOOL;
	ControlPower1: BOOL;
	ControlPower2: BOOL;
	Force_TipChange: BOOL;
	TipChange_Complete: BOOL;
	Reset_ChangeCount: BOOL;
	Enable_Dry_Cycle: BOOL;
	Local_DryCycle_Enables: UDINT;
	QA_Request_LH: BOOL;
	QA_Request_RH: BOOL;
	QA_Reinsert_LH: BOOL;
	QA_Reinsert_RH: BOOL;
	QA_Reset: UINT;
	QA_NOK_BinCount_Resets: UINT;	
	QA_NOK_Consecutive_Resets: UINT;
	
	Global_Robot_Speed: BYTE;
	Low_Speed_Req: BOOL;
	Force_Master_Test: BOOL;
	Force_Brake_Test: BOOL;
	Bypass_REQS: UDINT;
	CustomApplication_REQS: UDINT;
	Rxx_ToolChange_REQS: UDINT;
	T1_Zone_Test: BOOL;
	Production_Report_Trigger_ACKS: UDINT;
	Product_Report_Trigger_ACKS: UDINT;

	(*Sealer Related Bits*)
	SL01_Purge_REQS: UINT;
	SL02_Purge_REQS: UINT;
	SL03_Purge_REQS: UINT;
	SL04_Purge_REQS: UINT;
	SL01_Dispense_Bypass: UINT;
	SL02_Dispense_Bypass: UINT;
	SL03_Dispense_Bypass: UINT;
	SL04_Dispense_Bypass: UINT;



(*Standard UI Control For Operator Stations and Status of TWCAT Driver Sheet Comms*)
	(*IC01*)
	IC01_Requests: INT;				(*Bit 1 = Production, 2 = Materials, 3 = Maintenance*)
	IC01_COMM_STAT: INT;			(*Communication Status of Twincat driver sheet in Indusoft*)
	(*IC02*)
	IC02_Requests: INT;				(*Bit 1 = Production, 2 = Materials, 3 = Maintenance*)
	IC02_COMM_STAT: INT;			(*Communication Status of Twincat driver sheet in Indusoft*)
	(*IC03*)
	IC03_Requests: INT;				(*Bit 1 = Production, 2 = Materials, 3 = Maintenance*)
	IC03_COMM_STAT: INT;			(*Communication Status of Twincat driver sheet in Indusoft*)
	(*IC04*)
	IC04_Requests: INT;				(*Bit 1 = Production, 2 = Materials, 3 = Maintenance*)
	IC04_COMM_STAT: INT;			(*Communication Status of Twincat driver sheet in Indusoft*)
	(*IC05*)
	IC05_Requests: INT;				(*Bit 1 = Production, 2 = Materials, 3 = Maintenance*)
	IC05_COMM_STAT: INT;			(*Communication Status of Twincat driver sheet in Indusoft*)
	(*IC06*)
	IC06_Requests: INT;				(*Bit 1 = Production, 2 = Materials, 3 = Maintenance*)
	IC06_COMM_STAT: INT;			(*Communication Status of Twincat driver sheet in Indusoft*)
	(*IC07*)
	IC07_Requests: INT;				(*Bit 1 = Production, 2 = Materials, 3 = Maintenance*)
	IC07_COMM_STAT: INT;			(*Communication Status of Twincat driver sheet in Indusoft*)
	(*IC08*)
	IC08_Requests: INT;				(*Bit 1 = Production, 2 = Materials, 3 = Maintenance*)
	IC08_COMM_STAT: INT;			(*Communication Status of Twincat driver sheet in Indusoft*)

(*Specific Inputs from UI*)
	(*Robot Control*)
	Rxx_Weld_Inhibit: BOOL;
	Rxx_Dress_Req: BOOL;
	Rxx_TraccTCP_Req: BOOL;
	R1_Weld_Inhibit: BOOL;
	R1_Disable_Power: BOOL;
	R1_Temp_Start: BOOL;
	R1_Dress_Req: BOOL;
	R1_TraccTCP_Req: BOOL;
	R2_Weld_Inhibit: BOOL;
	R2_Disable_Power: BOOL;
	R2_Temp_Start: BOOL;
	R2_Dress_Req: BOOL;
	R2_TraccTCP_Req: BOOL;
	R3_Weld_Inhibit: BOOL;
	R3_Disable_Power: BOOL;
	R3_Temp_Start: BOOL;
	R3_Dress_Req: BOOL;
	R3_TraccTCP_Req: BOOL;
	R4_Weld_Inhibit: BOOL;
	R4_Disable_Power: BOOL;
	R4_Temp_Start: BOOL;
	R4_Dress_Req: BOOL;
	R4_TraccTCP_Req: BOOL;
	R5_Weld_Inhibit: BOOL;
	R5_Disable_Power: BOOL;
	R5_Temp_Start: BOOL;
	R5_Dress_Req: BOOL;
	R5_TraccTCP_Req: BOOL;
	R6_Weld_Inhibit: BOOL;
	R6_Disable_Power: BOOL;
	R6_Temp_Start: BOOL;
	R6_Dress_Req: BOOL;
	R6_TraccTCP_Req: BOOL;
	R7_Weld_Inhibit: BOOL;
	R7_Disable_Power: BOOL;
	R7_Temp_Start: BOOL;
	R7_Dress_Req: BOOL;
	R7_TraccTCP_Req: BOOL;
	R8_Weld_Inhibit: BOOL;
	R8_Disable_Power: BOOL;
	R8_Temp_Start: BOOL;
	R8_Dress_Req: BOOL;
	R8_TraccTCP_Req: BOOL;
	R9_Weld_Inhibit: BOOL;
	R9_Disable_Power: BOOL;
	R9_Temp_Start: BOOL;
	R9_Dress_Req: BOOL;
	R9_TraccTCP_Req: BOOL;
	R10_Weld_Inhibit: BOOL;
	R10_Disable_Power: BOOL;
	R10_Temp_Start: BOOL;
	R10_Dress_Req: BOOL;
	R10_TraccTCP_Req: BOOL;
	R11_Weld_Inhibit: BOOL;
	R11_Disable_Power: BOOL;
	R11_Temp_Start: BOOL;
	R11_Dress_Req: BOOL;
	R11_TraccTCP_Req: BOOL;
	R12_Weld_Inhibit: BOOL;
	R12_Disable_Power: BOOL;
	R12_Temp_Start: BOOL;
	R12_Dress_Req: BOOL;
	R12_TraccTCP_Req: BOOL;
	R13_Weld_Inhibit: BOOL;
	R13_Disable_Power: BOOL;
	R13_Temp_Start: BOOL;
	R13_Dress_Req: BOOL;
	R13_TraccTCP_Req: BOOL;
	R14_Weld_Inhibit: BOOL;
	R14_Disable_Power: BOOL;
	R14_Temp_Start: BOOL;
	R14_Dress_Req: BOOL;
	R14_TraccTCP_Req: BOOL;
	R15_Weld_Inhibit: BOOL;
	R15_Disable_Power: BOOL;
	R15_Temp_Start: BOOL;
	R15_Dress_Req: BOOL;
	R15_TraccTCP_Req: BOOL;
	R16_Weld_Inhibit: BOOL;
	R16_Disable_Power: BOOL;
	R16_Temp_Start: BOOL;
	R16_Dress_Req: BOOL;
	R16_TraccTCP_Req: BOOL;
	R17_Weld_Inhibit: BOOL;
	R17_Disable_Power: BOOL;
	R17_Temp_Start: BOOL;
	R17_Dress_Req: BOOL;
	R17_TraccTCP_Req: BOOL;
	R18_Weld_Inhibit: BOOL;
	R18_Disable_Power: BOOL;
	R18_Temp_Start: BOOL;
	R18_Dress_Req: BOOL;
	R18_TraccTCP_Req: BOOL;
	R19_Weld_Inhibit: BOOL;
	R19_Disable_Power: BOOL;
	R19_Temp_Start: BOOL;
	R19_Dress_Req: BOOL;
	R19_TraccTCP_Req: BOOL;
	R20_Weld_Inhibit: BOOL;
	R20_Disable_Power: BOOL;
	R20_Temp_Start: BOOL;
	R20_Dress_Req: BOOL;
	R20_TraccTCP_Req: BOOL;
	R21_Weld_Inhibit: BOOL;
	R21_Disable_Power: BOOL;
	R21_Temp_Start: BOOL;
	R21_Dress_Req: BOOL;
	R21_TraccTCP_Req: BOOL;
	R22_Weld_Inhibit: BOOL;
	R22_Disable_Power: BOOL;
	R22_Temp_Start: BOOL;
	R22_Dress_Req: BOOL;
	R22_TraccTCP_Req: BOOL;
	R23_Weld_Inhibit: BOOL;
	R23_Disable_Power: BOOL;
	R23_Temp_Start: BOOL;
	R23_Dress_Req: BOOL;
	R23_TraccTCP_Req: BOOL;
	R24_Weld_Inhibit: BOOL;
	R24_Disable_Power: BOOL;
	R24_Temp_Start: BOOL;
	R24_Dress_Req: BOOL;
	R24_TraccTCP_Req: BOOL;
	R25_Weld_Inhibit: BOOL;
	R25_Disable_Power: BOOL;
	R25_Temp_Start: BOOL;
	R25_Dress_Req: BOOL;
	R25_TraccTCP_Req: BOOL;
	R26_Weld_Inhibit: BOOL;
	R26_Disable_Power: BOOL;
	R26_Temp_Start: BOOL;
	R26_Dress_Req: BOOL;
	R26_TraccTCP_Req: BOOL;
	R27_Weld_Inhibit: BOOL;
	R27_Disable_Power: BOOL;
	R27_Temp_Start: BOOL;
	R27_Dress_Req: BOOL;
	R27_TraccTCP_Req: BOOL;
	R28_Weld_Inhibit: BOOL;
	R28_Disable_Power: BOOL;
	R28_Temp_Start: BOOL;
	R28_Dress_Req: BOOL;
	R28_TraccTCP_Req: BOOL;
	R29_Weld_Inhibit: BOOL;
	R29_Disable_Power: BOOL;
	R29_Temp_Start: BOOL;
	R29_Dress_Req: BOOL;
	R29_TraccTCP_Req: BOOL;
	R30_Weld_Inhibit: BOOL;
	R30_Disable_Power: BOOL;
	R30_Temp_Start: BOOL;
	R30_Dress_Req: BOOL;
	R30_TraccTCP_Req: BOOL;

	(*Fixture Control*)
	Fix01_Discrete_In: udt_FixXX_Input_Image_20180202;
	Fix02_Discrete_In: udt_FixXX_Input_Image_20180202;
	Fix03_Discrete_In: udt_FixXX_Input_Image_20180202;
	Fix04_Discrete_In: udt_FixXX_Input_Image_20180202;
	Fix05_Discrete_In: udt_FixXX_Input_Image_20180202;
	Fix06_Discrete_In: udt_FixXX_Input_Image_20180202;
	Fix07_Discrete_In: udt_FixXX_Input_Image_20180202;
	Fix08_Discrete_In: udt_FixXX_Input_Image_20180202;
	Fix09_Discrete_In: udt_FixXX_Input_Image_20180202;
	Fix10_Discrete_In: udt_FixXX_Input_Image_20180202;
	Fix11_Discrete_In: udt_FixXX_Input_Image_20180202;
	Fix12_Discrete_In: udt_FixXX_Input_Image_20180202;
	Fix13_Discrete_In: udt_FixXX_Input_Image_20180202;
	Fix14_Discrete_In: udt_FixXX_Input_Image_20180202;
	Fix15_Discrete_In: udt_FixXX_Input_Image_20180202;
	Fix16_Discrete_In: udt_FixXX_Input_Image_20180202;

	Fix101_Discrete_In: udt_FixXX_Input_Image_20180202;
	Fix102_Discrete_In: udt_FixXX_Input_Image_20180202;
	Fix103_Discrete_In: udt_FixXX_Input_Image_20180202;
	Fix104_Discrete_In: udt_FixXX_Input_Image_20180202;
	Fix105_Discrete_In: udt_FixXX_Input_Image_20180202;
	Fix106_Discrete_In: udt_FixXX_Input_Image_20180202;
	Fix107_Discrete_In: udt_FixXX_Input_Image_20180202;
	Fix108_Discrete_In: udt_FixXX_Input_Image_20180202;
	Fix109_Discrete_In: udt_FixXX_Input_Image_20180202;
	Fix110_Discrete_In: udt_FixXX_Input_Image_20180202;
	Fix111_Discrete_In: udt_FixXX_Input_Image_20180202;
	Fix112_Discrete_In: udt_FixXX_Input_Image_20180202;

	(*Nut Weld based LVDTs*)
	NutWeld_LVDT_Discrete_In: ARRAY [0..5] OF udt_NutWeldLVDT_Input_Image_20250616;
	
	(*Custom addition for SIC marking units*)
	SIC01_BypassReq: BOOL;
	SIC02_BypassReq: BOOL;


	(*Generic Servo Control*)
	SD: ARRAY [0..30] OF udt_SDxx_FromUI_20220224;
	
	(*IV2/3 UI Inputs*)
	IVx_Discrete_In: ARRAY [0..5] OF udt_IVxx_Input_Image_20250812;
	
	(*SRxx*)
	SRx_Discrete_In : ARRAY [0..1] OF udt_SRxx_Input_Image;	

	END_STRUCT
END_TYPE

// ---- Data types/UI udts/udt_UIcommon_Output_20251008.TcDUT
(*udt (user defined type) for interfacing to UI (User Interface)
this udt represents data that is passed from PLC to ALL UIs

	Author(S): Rob Remillard/Brent Lekx-Toniolo of Sodecia GTAC;
	Version 1.0 (Named udt_HMI_Output): August 2010
		- Initial Concept
	Version 20141014
		- Increase for 30 Robot framework + Fix Renaming, b.lekx-toniolo
	Version 20141128
		- Added ESW Count Option, b.lekx-toniolo
		- Added More WSxxs, b.lekx-toniolo
	Version 20141209
		- Added TTxx Ints for location indexes of Turntables, b.lekx-toniolo
	Version 20141211
		- Added SMB Image, b.lekx-toniolo
		- Updated Ecat Master Instance, b.lekx-toniolo
	Version 20150226
		- Added Target Cycle Time for display on UI screen(s), b.lekx-toniolo
	Version 20150812
		- Added PD Count for display on UI screen(s), b.lekx-toniolo
	Version 20150827
		- Renamed Option_HumanFix_Count to Option_HumanFix_Enables, b.lekx-toniolo
	Version 20160113
		- Increased fault area size and added area for water setpoint options, b.lekx-toniolo
		- Added UI Prompt flags for controls faults prompting , b.lekx-toniolo
	Version 20160418
		- Added Area for Robot Water Flow Timeout feature configuration data, b.lekx-toniolo
		- updated ECAT Master area to include new new image with HW config data, b.lekx-toniolo 
	Version 20160519
		-Added udts for Each Shift Structure Configuration, b.lekx-toniolo
		- Removed Old Model Change Allow Bools, b.lekx-toniolo
		- Added Report_Trigger_Acks, b.lekx-toniolo
		- Added Rxx_ToolChange_Acks, b.lekx-toniolo
	Version 20161129
		-Custom setup for SIC marking, RRemillard	
	Version 20161206
		-added sealer bits, j.vandongen
	Version 20170626
		- added local dry cycle, b.lekx-toniolo / c.drees (edge automation)
	Version 20170801
		-added bit to control monitoring spaces from plc, RRemillard
	Version 20170804
		-added cycle hold ack, j.vandongen
	Version 20180417	
		-added Option_EOAT_Count, j.vandongen
		-added Option_LaserController, j.vandongen
		-changed var type Config_Fault, j.vandongen
		-added EOAT discrete images, j.vandongen
		-added SD option count, j.vandongen
	Version 20191125
		- Added ProdConfig_Common, b.lekx-toniolo 
		- Update names for EOAT -> UI interface to correct naming mismatch in UI driver sheet, b.lekx-toniolo
	Version 20191210
		-Added Code to deal with TC3 Changes:
			-Motherboard data is no longer a device in the I/O tree and MUST be read in from the MDP.  Not all data is available anymore, so UDT modified
				to show data changes
			-Application data is no longer stored in the same global system variable as before, new structure added for the App data
			-Task Data is no longer stored in the same global system variable as before, new strucuture added for the task data.
	Version 20220224
		- Overhaul during TcUI migration project, b.lekx-toniolo / c.drees
		- Added in In_Sim_Mode for integration into simulation, b.lekx-toniolo	
	Version 20240909
		- Increased Product Report Data Area to give EOATs a storage location, b.lekx-toniolo	
	Version 20240926
		- Added in data area for MDxx (Motorized Door) component, b.lekx-toniolo	
	Version 20241121
		- PD to IS rename, as per GH SSCC610 repo Issue#162, b.lekx-toniolo
	Version 20250616
		- Added in Nut Weld Based LVDT Output Image, b.lekx-toniolo	
	Version 20250716
		- Added in Exceed_Counter_Value, per SSCC610 GH Issue #235, b.lekx-toniolo
	Version 20250723
		- Added in config count and general discrete images for VFD additions, b.lekx-toniolo / r. jones
	Version20251008
		- MDxx instance update, b.lekx-toniolo	
*)

TYPE udt_UIcommon_Output_20251008 :
	STRUCT
(*Configuration Data to UI*)
	Machine_Serial: STRING;
	Machine_Common_Name: STRING;
	Machine_Build_Used: STRING;
	Machine_Appl_Dev: STRING;
	
	ProdConfig_Target_CycleTime: TIME;

	ProdConfig_Common: udt_Generic_ShiftCommonConfig_20220420;
	ProdConfig_Day: udt_Generic_ShiftConfigUDINT_20160531;
	ProdConfig_Aft: udt_Generic_ShiftConfigUDINT_20160531;
	ProdConfig_Mid: udt_Generic_ShiftConfigUDINT_20160531;

	Option_Air1: BOOL;
	Option_Air2: BOOL;
	Option_Water1: BOOL;
	Option_Water2: BOOL;

	Option_WaterTimeOut_Enable: BOOL;
	Option_WaterFlowTimeOut_SP: TIME;
	Option_WaterTempHighLimit1: REAL;
	Option_WaterFlowLowLimit1: REAL;
	Option_WaterTempHighLimit2: REAL;
	Option_WaterFlowLowLimit2: REAL;

	Option_IS_Count: UINT;
	Option_ESW_Count: UINT;
	Option_MD_Count: UINT;
	Option_IC_Count: UINT;
	Option_HumanFix_Enables: UDINT;
	Option_InternalFix_Count: UINT;
	Option_Robot_Count: UINT;
	Option_Ped_Count: UINT;
	Option_StudController_Count: UINT;
	Option_SealController_Count: UINT;
	Option_NutWelder_Count: UINT;
	Option_EOAT_Count: UINT;
	Option_LaserController_Count: UINT;
	Option_SD_Count: UINT;
	Option_VFD_Count: UINT;
	Config_Fault:UDINT;

(*Standard Outputs to UI*)
	(*Common to Cell*)
	ControlPower1_OK: BOOL; (*Control Power is ON*)
	ControlPower2_OK: BOOL;	(*spare*)
	CycleHold_OK: BOOL;
	Estops_OK: BOOL;		(*All Estops OK and Reset*)
	Safety_Gates_OK: BOOL;	(*All Safety Gates OK and Reset*)
	Faults_OK: BOOL;		(*No Major Faults*)
	TipChangeReq_OK: BOOL;
	TipChangeComp_OK: BOOL;
	Change_Count: INT;
	TipChange_Part_Count: INT;
	InDryCycle:BOOL;
	In_Local_DryCycle:UDINT;
	Allow_Model_Change: BOOL;
	QA_LH_Ready: BOOL;
	QA_RH_Ready: BOOL;
	QA_NOK_BinCounts: ARRAY [0..16] OF UINT;
	Spare1: BOOL;
	Spare2: BOOL;
	SMB_Status_Image: udt_SMB_Status_20141211;
	EtherCat_Master_Image: udt_ECATMaster_Image_20220224;
	EL6900_FB_Errors1: DINT;
	EL6900_Comm_Errors1: DINT;
	EL6900_Out_Errors1: DINT;
	EL6900_FB_Errors2: DINT;
	EL6900_Comm_Errors2: DINT;
	EL6900_Out_Errors2: DINT;
	Overall_Controls_Fault: UINT;
	In_Low_Speed: BOOL;
	Under_Construction: BOOL;	(*System is Under Construction*)
	In_Sim_Mode: BOOL; 			(*System in Simulation mode, added during project 90034*)
	MasterTest_Req_OK: BOOL;
	BrakeTest_Req_OK: BOOL;
	Rxx_ReadyFor_TipChange: UDINT;
	Bypass_ACKS: UDINT;
	CustomApplication_ACKS: UDINT;
	Rxx_ToolChange_ACKS: UDINT;
	T1_Zone_Test_ACK: BOOL;
	Production_Report_Trigger_REQS: UDINT;
	Product_Report_Trigger_REQS: UDINT;

	(* TC3 Specific data types for App data, Task data and Motherboard Diagnostics *)
	Appdata 	:PlcAppSystemInfo;
	TaskData	:PlcTaskSystemInfo;
	MboardData	:udt_HardwareDiags;
	Exceed_Counter_Value: UDINT;
	
	(*Sealer Bits*)
	SL01_Dispense_Count: UINT;
	SL02_Dispense_Count: UINT;
	SL03_Dispense_Count: UINT;
	SL04_Dispense_Count: UINT;
	SL01_Bypass_ACK: UINT;
	SL02_Bypass_ACK: UINT;
	SL03_Bypass_ACK: UINT;
	SL04_Bypass_ACK: UINT;


(*Standard UI Visualization For Operator Stations*)
	(*IC01*)
	IC01OP1_LCHVR: BOOL;
	IC01OP1_LCHHR: BOOL;
	IC01OP1_LCRVR: BOOL;
	IC01OP2_LCHVR: BOOL;
	IC01OP2_LCHHR: BOOL;
	IC01OP2_LCRVR: BOOL;
	(*IC02*)
	IC02OP1_LCHVR: BOOL;
	IC02OP1_LCHHR: BOOL;
	IC02OP1_LCRVR: BOOL;
	IC02OP2_LCHVR: BOOL;
	IC02OP2_LCHHR: BOOL;
	IC02OP2_LCRVR: BOOL;
	(*IC03*)
	IC03OP1_LCHVR: BOOL;
	IC03OP1_LCHHR: BOOL;
	IC03OP1_LCRVR: BOOL;
	IC03OP2_LCHVR: BOOL;
	IC03OP2_LCHHR: BOOL;
	IC03OP2_LCRVR: BOOL;
	(*IC04*)
	IC04OP1_LCHVR: BOOL;
	IC04OP1_LCHHR: BOOL;
	IC04OP1_LCRVR: BOOL;
	IC04OP2_LCHVR: BOOL;
	IC04OP2_LCHHR: BOOL;
	IC04OP2_LCRVR: BOOL;
	(*IC05*)
	IC05OP1_LCHVR: BOOL;
	IC05OP1_LCHHR: BOOL;
	IC05OP1_LCRVR: BOOL;
	IC05OP2_LCHVR: BOOL;
	IC05OP2_LCHHR: BOOL;
	IC05OP2_LCRVR: BOOL;
	(*IC06*)
	IC06OP1_LCHVR: BOOL;
	IC06OP1_LCHHR: BOOL;
	IC06OP1_LCRVR: BOOL;
	IC06OP2_LCHVR: BOOL;
	IC06OP2_LCHHR: BOOL;
	IC06OP2_LCRVR: BOOL;
	(*IC07*)
	IC07OP1_LCHVR: BOOL;
	IC07OP1_LCHHR: BOOL;
	IC07OP1_LCRVR: BOOL;
	IC07OP2_LCHVR: BOOL;
	IC07OP2_LCHHR: BOOL;
	IC07OP2_LCRVR: BOOL;
	(*IC08*)
	IC08OP1_LCHVR: BOOL;
	IC08OP1_LCHHR: BOOL;
	IC08OP1_LCRVR: BOOL;
	IC08OP2_LCHVR: BOOL;
	IC08OP2_LCHHR: BOOL;
	IC08OP2_LCRVR: BOOL;


	(*Location Index for Animation of Turntables*)
	TT01_Location_Index: INT;
	TT02_Location_Index: INT;
	TT03_Location_Index: INT;
	TT04_Location_Index: INT;
	TT05_Location_Index: INT;
	TT06_Location_Index: INT;
	TT07_Location_Index: INT;
	TT08_Location_Index: INT;
	TT09_Location_Index: INT;

	(*Fixture Visualization*)
	Fix01_Discrete_Image: udt_FixXX_Output_Image_20250721_CUSTOM;
	Fix02_Discrete_Image: udt_FixXX_Output_Image_20250721_CUSTOM;
	Fix03_Discrete_Image: udt_FixXX_Output_Image_20220715;
	Fix04_Discrete_Image: udt_FixXX_Output_Image_20220715;
	Fix05_Discrete_Image: udt_FixXX_Output_Image_20220715;
	Fix06_Discrete_Image: udt_FixXX_Output_Image_20220715;
	Fix07_Discrete_Image: udt_FixXX_Output_Image_20220715;
	Fix08_Discrete_Image: udt_FixXX_Output_Image_20220715;
	Fix09_Discrete_Image: udt_FixXX_Output_Image_20220715;
	Fix10_Discrete_Image: udt_FixXX_Output_Image_20220715;
	Fix11_Discrete_Image: udt_FixXX_Output_Image_20220715;
	Fix12_Discrete_Image: udt_FixXX_Output_Image_20220715;
	Fix13_Discrete_Image: udt_FixXX_Output_Image_20220715;
	Fix14_Discrete_Image: udt_FixXX_Output_Image_20220715;
	Fix15_Discrete_Image: udt_FixXX_Output_Image_20220715;
	Fix16_Discrete_Image: udt_FixXX_Output_Image_20220715;

	Fix101_Discrete_Image: udt_FixXX_Output_Image_20220715;
	Fix102_Discrete_Image: udt_FixXX_Output_Image_20220715;
	Fix103_Discrete_Image: udt_FixXX_Output_Image_20220715;
	Fix104_Discrete_Image: udt_FixXX_Output_Image_20220715;
	Fix105_Discrete_Image: udt_FixXX_Output_Image_20220715;
	Fix106_Discrete_Image: udt_FixXX_Output_Image_20220715;
	Fix107_Discrete_Image: udt_FixXX_Output_Image_20220715;
	Fix108_Discrete_Image: udt_FixXX_Output_Image_20220715;
	Fix109_Discrete_Image: udt_FixXX_Output_Image_20220715;
	Fix110_Discrete_Image: udt_FixXX_Output_Image_20220715;
	Fix111_Discrete_Image: udt_FixXX_Output_Image_20220715;
	Fix112_Discrete_Image: udt_FixXX_Output_Image_20220715;

	(*End of Arm Tooling Visualization*)
	EOAT01_Discrete_Image: udt_EOATxx_Image_20170607;
	EOAT02_Discrete_Image: udt_EOATxx_Image_20170607;
	EOAT03_Discrete_Image: udt_EOATxx_Image_20170607;
	EOAT04_Discrete_Image: udt_EOATxx_Image_20170607;
	EOAT05_Discrete_Image: udt_EOATxx_Image_20170607;
	EOAT06_Discrete_Image: udt_EOATxx_Image_20170607;
	EOAT07_Discrete_Image: udt_EOATxx_Image_20170607;
	EOAT08_Discrete_Image: udt_EOATxx_Image_20170607;
	EOAT09_Discrete_Image: udt_EOATxx_Image_20170607;
	EOAT10_Discrete_Image: udt_EOATxx_Image_20170607;

	(*Nut Weld based LVDTs*)
	NutWeld_LVDT_Discrete_Image: ARRAY [0..5] OF udt_NutWeldLVDT_Output_Image_20250616;

	(*Standard GTAC Component I/O Visualization*)
	(*ISxx*)
	IS: ARRAY [0..1] OF udt_ISxx_ToUI_20241121;
	(*ICxx*)
	IC: ARRAY [0..8] OF udt_ICxx_ToUI_20220224;
	(*Rxx*)
	Robot: ARRAY [0..30] OF udt_Rxx_ToUI_20220224;
	(*SSxx*)
	SS: ARRAY [0..2] OF udt_SSxx_ToUI_20250704;
	(*STxx*)
	Stud: ARRAY [0..10] OF udt_STxx_ToUI_20220224;
	(*SLxx*)
	SL: ARRAY [0..10] OF udt_SLxx_ToUI_20220224;
	(*SDxx*)
	SD: ARRAY [0..30] OF udt_SDxx_ToUI_20220224;
	(*NWxx*)
	NW: ARRAY [0..5] OF udt_NWxx_ToUI_20220224;
	(*ESWxx*)
	ESW: ARRAY [0..4] OF udt_ESWxx_ToUI_20220224;
	(*LSRxx*)
	LSR: ARRAY [0..9] OF udt_LSRxx_ToUI_20220224;
	(*PEDxx*)
	PED: ARRAY[0..30] OF udt_PEDxx_Image_20240808;
	(*MDxx*)
	MD: ARRAY[0..5] OF udt_MDxx_ToUI_20251008;
	(*VFDxx*)
	VFD: ARRAY[0..5] OF udt_VFDxx_ToUI_20250723;
	(*IV2/3xx*)
	IVx: ARRAY [0..5] OF udt_IVxx_ToUI_20250808;
	(*Smart Ray*)
	SRx: ARRAY [0..1] OF udt_SRxx_ToUI_20260122;	
	
	(*Production Report Fix XX*)
	(*Elements 1 - 16 -> Fix01 - Fix16*)
	ProdReport: ARRAY [0..16] OF udt_ProdReportxx_ToUI_20220224;
	
	(*Product Reports Fix XX*)
	(*Element 0 -> Blank (intentionally)*)
	(*Elements 1 - 16 -> Fix01 - Fix16*)
	(*Elements 17 - 28 -> Fix101 - Fix112*)
	(*Elements 31 - 40 -> EOAT01 - EOAT10*)
	ProductReport: ARRAY [0..40] OF udt_Generic_ProductReportData_20240909;
		
	
	(*System Faults*)
	System_Faults: ARRAY[0..1639] OF BOOL:=[ FALSE]; (*General System Faults*)
	(*Component Controls Fault Flag for Prompting on UI*)
	ICxx_UI_FaultPrompts: UDINT;
	Rxx_UI_FaultPrompts: UDINT;
	Rxx_UI_FaultPrompts_2: UDINT;
	ISxx_UI_FaultPrompts: UDINT;
	SDxx_UI_FaultPrompts: UDINT;
	STxx_UI_FaultPrompts: UDINT;
	SLxx_UI_FaultPrompts: UDINT;
	NWxx_UI_FaultPrompts: UDINT;
	MDxx_UI_FaultPrompts: UDINT;
	VFDxx_UI_FaultPrompts: UDINT;
	MISCxx_UI_FaultPrompts: UDINT;

	(*Custom Items for one time SIC Marker install*)
	SIC01_DpState: INT;
	SIC01_ProfinodeOK: BOOL;
	SIC01_Running: BOOL;
	SIC01_LastDot: BOOL;
	SIC01_BackHome: BOOL;
	SIC01_Complete: BOOL;
	SIC01_Reply: STRING;

	SIC02_DpState: INT;
	SIC02_ProfinodeOK: BOOL;
	SIC02_Running: BOOL;
	SIC02_LastDot: BOOL;
	SIC02_BackHome: BOOL;
	SIC02_Complete: BOOL;
	SIC02_Reply: STRING;

	END_STRUCT
END_TYPE

// ---- Global Variables/Global_Persistent_Variables.TcGVL
{attribute 'Tc2GvlVarNames'}
VAR_GLOBAL PERSISTENT

	(* Persistent Data Frame Work for Interface to UI(s), be sure to see "Work Space" in Resources Tab for entitiy export*)
	(*Interfacing to all UI(s)*)
		In_From_ICxx_Pers: udt_UIcommon_InputPers_20250612; (* Data Frame Work for Receiving Persistent Data from any IC*)

		
	(*Part Data Area Custom for this machine - See "Product_Tracking" Action Under Main*)
	(* 
		The Generic_PassFail_Notes variable will be used for tracking state of each fixture the part visits
		
		Valid values will be:
			"Pass" = Inspection of part complete and is considered passed or OK
			"Fail" = Inspection of part is complete and is considered failed or NOK
			"Comp" = The required Task has been completed
			Blank =	The required Task has not yet been completed
			
		Array Layout to track above will be:
			[1] = Fix01 (Set to "Comp" when welding is complete)
			[2] = Fix02 (Set to "Comp" when welding is complete)
	
			[3] = Fix03 (Set to "Comp" when welding is complete)
			[4] = Fix04 (Set to "Comp" when welding is complete)
			
			[5] = Fix05 (Set to "Comp" when insertion of part is ready)
	
			[11] = Fix101 (Set to "Comp" when welding is complete)
			
			[12] = Fix102 (Set to "Pass" or "Fail" depending on inspection results)
			[13] = Fix103 (Set to "Comp" when part is successfully placed on conveyor to QA / NOK)
			[15] = Fix105 (Set to "Comp" when part is successfully placed on conveyor to Paint)

	*)	
	
	Blank_ProductData_Pers: udt_Generic_ProductReportData_20240909;		(*Blank data area used for blanking / resetting purposes*)
	
	Fix01_ProductData_Pers: udt_Generic_ProductReportData_20240909;		(*First Geo Set on TT01*)
	Fix02_ProductData_Pers: udt_Generic_ProductReportData_20240909;		(*First Geo Set on TT01*)

	EOAT04_1_ProductData_Pers: udt_Generic_ProductReportData_20240909;	(*MH Robot EOAT Side 1*)
	EOAT04_2_ProductData_Pers: udt_Generic_ProductReportData_20240909;	(*MH Robot EOAT Side 2*)
	Fix101_ProductData_Pers: udt_Generic_ProductReportData_20240909;	(*Finishing first Geo sets*)
	
	Fix03_ProductData_Pers: udt_Generic_ProductReportData_20240909;		(*Second Geo and Finish on TT02*)
	Fix04_ProductData_Pers: udt_Generic_ProductReportData_20240909;		(*Second Geo and Finish on TT02*)

	
	Fix102_ProductData_Pers: udt_Generic_ProductReportData_20240909;	(*Vision Inspection Station*)
	
	Fix05_ProductData_Pers: udt_Generic_ProductReportData_20240909;		(*Insert Rewroked Parts Fixture (Insert parts only)*)

	Fix103_ProductData_Pers: udt_Generic_ProductReportData_20240909;	(*QA Request / First off part / NOK (offload parts only)*)
	
	Fix104_ProductData_Pers: ARRAY [0..5] OF udt_Generic_ProductReportData_20240909;	(*Buffer rack before Paint (used if paint goes down*)
	
	Fix105_ProductData_Pers: udt_Generic_ProductReportData_20240909;	(*Hanging Rack to Paint*)
	
	
END_VAR

// ---- Global Variables/Global_Variables.TcGVL
{attribute 'Tc2GvlVarNames'}
VAR_GLOBAL
(*Modify This Record To Customize Each Robot Work Area, See Task ID Record Program*)

		(*All Task IDs*)
		Dropoff_Fix01: UINT;
		Weld_Fix01: UINT;
		Pickup_Fix01: UINT;
		Seal_Fix01: UINT;
		Stud_Fix01: UINT;
		Sweep_Fix01: UINT;

		Dropoff_Fix02: UINT;
		Weld_Fix02: UINT;
		Pickup_Fix02: UINT;
		Seal_Fix02: UINT;
		Stud_Fix02: UINT;
		Sweep_Fix02: UINT;

		Dropoff_Fix03: UINT;
		Weld_Fix03: UINT;
		Pickup_Fix03: UINT;
		Seal_Fix03: UINT;
		Stud_Fix03: UINT;
		Sweep_Fix03: UINT;

		Dropoff_Fix04: UINT;
		Weld_Fix04: UINT;
		Pickup_Fix04: UINT;
		Seal_Fix04: UINT;
		Stud_Fix04: UINT;
		Sweep_Fix04: UINT;

		Dropoff_Fix05: UINT;
		Weld_Fix05: UINT;
		Pickup_Fix05: UINT;
		Seal_Fix05: UINT;
		Stud_Fix05: UINT;
		Sweep_Fix05: UINT;

		Dropoff_Fix06: UINT;
		Weld_Fix06: UINT;
		Pickup_Fix06: UINT;
		Seal_Fix06: UINT;
		Stud_Fix06: UINT;
		Sweep_Fix06: UINT;

		Dropoff_Fix07: UINT;
		Weld_Fix07: UINT;
		Pickup_Fix07: UINT;
		Seal_Fix07: UINT;
		Stud_Fix07: UINT;
		Sweep_Fix07: UINT;

		Dropoff_Fix08: UINT;
		Weld_Fix08: UINT;
		Pickup_Fix08: UINT;
		Seal_Fix08: UINT;
		Stud_Fix08: UINT;
		Sweep_Fix08: UINT;

		Dropoff_Fix09: UINT;
		Weld_Fix09: UINT;
		Pickup_Fix09: UINT;
		Seal_Fix09: UINT;
		Stud_Fix09: UINT;
		Sweep_Fix09: UINT;

		Dropoff_Fix10: UINT;
		Weld_Fix10: UINT;
		Pickup_Fix10: UINT;
		Seal_Fix10: UINT;
		Stud_Fix10: UINT;
		Sweep_Fix10: UINT;

		Dropoff_Fix11: UINT;
		Weld_Fix11: UINT;
		Pickup_Fix11: UINT;
		Seal_Fix11: UINT;
		Stud_Fix11: UINT;
		Sweep_Fix11: UINT;

		Dropoff_Fix12: UINT;
		Weld_Fix12: UINT;
		Pickup_Fix12: UINT;
		Seal_Fix12: UINT;
		Stud_Fix12: UINT;
		Sweep_Fix12: UINT;

		Dropoff_Fix13: UINT;
		Weld_Fix13: UINT;
		Pickup_Fix13: UINT;
		Seal_Fix13: UINT;
		Stud_Fix13: UINT;
		Sweep_Fix13: UINT;

		Dropoff_Fix14: UINT;
		Weld_Fix14: UINT;
		Pickup_Fix14: UINT;
		Seal_Fix14: UINT;
		Stud_Fix14: UINT;
		Sweep_Fix14: UINT;

		Dropoff_Fix15: UINT;
		Weld_Fix15: UINT;
		Pickup_Fix15: UINT;
		Seal_Fix15: UINT;
		Stud_Fix15: UINT;
		Sweep_Fix15: UINT;

		Dropoff_Fix16: UINT;
		Weld_Fix16: UINT;
		Pickup_Fix16: UINT;
		Seal_Fix16: UINT;
		Stud_Fix16: UINT;
		Sweep_Fix16: UINT;

		(*Tasks Associated with Entire Work Area*)
		Dropoff_Fix101: UINT;
		Weld_Fix101: UINT;
		Pickup_Fix101: UINT;
		Seal_Fix101: UINT;
		Stud_Fix101: UINT;
		Sweep_Fix101: UINT;

		Dropoff_Fix102: UINT;
		Weld_Fix102: UINT;
		Pickup_Fix102: UINT;
		Seal_Fix102: UINT;
		Stud_Fix102: UINT;
		Sweep_Fix102: UINT;

		Dropoff_Fix103: UINT;
		Weld_Fix103: UINT;
		Pickup_Fix103: UINT;
		Seal_Fix103: UINT;
		Stud_Fix103: UINT;
		Sweep_Fix103: UINT;

		Dropoff_Fix104: UINT;
		Weld_Fix104: UINT;
		Pickup_Fix104: UINT;
		Seal_Fix104: UINT;
		Stud_Fix104: UINT;
		Sweep_Fix104: UINT;

		Dropoff_Fix105: UINT;
		Weld_Fix105: UINT;
		Pickup_Fix105: UINT;
		Seal_Fix105: UINT;
		Stud_Fix105: UINT;
		Sweep_Fix105: UINT;

		Dropoff_Fix106: UINT;
		Weld_Fix106: UINT;
		Pickup_Fix106: UINT;
		Seal_Fix106: UINT;
		Stud_Fix106: UINT;
		Sweep_Fix106: UINT;

		Dropoff_Fix107: UINT;
		Weld_Fix107: UINT;
		Pickup_Fix107: UINT;
		Seal_Fix107: UINT;
		Stud_Fix107: UINT;
		Sweep_Fix107: UINT;

		Dropoff_Fix108: UINT;
		Weld_Fix108: UINT;
		Pickup_Fix108: UINT;
		Seal_Fix108: UINT;
		Stud_Fix108: UINT;
		Sweep_Fix108: UINT;

		Dropoff_Fix109: UINT;
		Weld_Fix109: UINT;
		Pickup_Fix109: UINT;
		Seal_Fix109: UINT;
		Stud_Fix109: UINT;
		Sweep_Fix109: UINT;

		Dropoff_Fix110: UINT;
		Weld_Fix110: UINT;
		Pickup_Fix110: UINT;
		Seal_Fix110: UINT;
		Stud_Fix110: UINT;
		Sweep_Fix110: UINT;

		Dropoff_Fix111: UINT;
		Weld_Fix111: UINT;
		Pickup_Fix111: UINT;
		Seal_Fix111: UINT;
		Stud_Fix111: UINT;
		Sweep_Fix111: UINT;

		Dropoff_Fix112: UINT;
		Weld_Fix112: UINT;
		Pickup_Fix112: UINT;
		Seal_Fix112: UINT;
		Stud_Fix112: UINT;
		Sweep_Fix112: UINT;

		Work_Ped01: UINT;
		Work_Ped02: UINT;
		Work_Ped03: UINT;
		Work_Ped04: UINT;
		Work_Ped05: UINT;
		Work_Ped06: UINT;
		Work_Ped07: UINT;
		Work_Ped08: UINT;
		Work_Ped09: UINT;
		Work_Ped10: UINT;
		Work_Ped11: UINT;
		Work_Ped12: UINT;
		Work_Ped13: UINT;
		Work_Ped14: UINT;
		Work_Ped15: UINT;
		Work_Ped16: UINT;
		Work_Ped17: UINT;
		Work_Ped18: UINT;
		Work_Ped19: UINT;
		Work_Ped20: UINT;
		Work_Ped21: UINT;
		Work_Ped22: UINT;
		Work_Ped23: UINT;
		Work_Ped24: UINT;
		Work_Ped25: UINT;
		Work_Ped26: UINT;
		Work_Ped27: UINT;
		Work_Ped28: UINT;
		Work_Ped29: UINT;
		Work_Ped30: UINT;

		Master_Test: UINT;
		Brake_Test: UINT;
		Tip_Dress: UINT;
		Tip_Change: UINT;
		Tip_Change_EXT: UINT;
		Tracc_Tcp: UINT;
		
		(*Robot Types*)
		MOTO_ERC: UINT;
		MOTO_MRC: UINT;
		MOTO_XRC: UINT;
		MOTO_NX100: UINT;
		MOTO_DX100: UINT;
		MOTO_DX100_Dual: UINT;
		MOTO_DX100_32: UINT;
		KUKA_KRC2: UINT;
		KUKA_KRC4: UINT;
		KUKA_KRC4_SAFEOP: UINT;
		KUKA_KRC4_SAFEOP_Small: UINT;
		KUKA_KRC4_SAFEOP_ATI: UINT;
		KUKA_KRC4c_SAFEOP_AGILUS: UINT;
		KUKA_KRC4_SAFEOP_TurnTable: UINT;

(*$$$$$$$$$$$$$$$$$$$$ Globally Scoped Data that Requires Write Access By All FBs and Progs $$$$$$$$$$$$$$$$$$$$$$$$$$$$*)
		Pulse_1S_FB: FB_Pulse_Generator;
		Pulse_1S: BOOL;
		Pulse_500ms_FB: FB_Pulse_Generator;
		Pulse_500ms: BOOL;
		Pulse_CoERead_FB: FB_Pulse_Generator;
		Pulse_CoERead: BOOL;

		(*Global Config Resets (See UI Prog for Mapping)*)
		ResetAllConfig_To_Default: BOOL;
		ResetProdConfig_To_Default: BOOL;

		(*Generic Data Frame Works*)
		R1_Data: udt_Generic_Robot_20161202;				(*Global Data Area for R01 Input*)
		R2_Data: udt_Generic_Robot_20161202;				(*Global Data Area for R02 Input*)
		R3_Data: udt_Generic_Robot_20161202;				(*Global Data Area for R03 Input*)
		R4_Data: udt_Generic_Robot_20250711_CUSTOM;				(*Global Data Area for R04 Input*)
		R5_Data: udt_Generic_Robot_20161202;				(*Global Data Area for R05 Input*)
		R6_Data: udt_Generic_Robot_20161202;				(*Global Data Area for R06 Input*)
		R7_Data: udt_Generic_Robot_20161202;				(*Global Data Area for R07 Input*)
		R8_Data: udt_Generic_Robot_20161202;				(*Global Data Area for R08 Input*)
		R9_Data: udt_Generic_Robot_20161202;				(*Global Data Area for R09 Input*)
		R10_Data: udt_Generic_Robot_20161202;				(*Global Data Area for R10 Input*)
		R11_Data: udt_Generic_Robot_20161202;				(*Global Data Area for R11 Input*)
		R12_Data: udt_Generic_Robot_20161202;				(*Global Data Area for R12 Input*)
		R13_Data: udt_Generic_Robot_20161202;				(*Global Data Area for R13 Input*)
		R14_Data: udt_Generic_Robot_20161202;				(*Global Data Area for R14 Input*)
		R15_Data: udt_Generic_Robot_20161202;				(*Global Data Area for R15 Input*)
		R16_Data: udt_Generic_Robot_20161202;				(*Global Data Area for R16 Input*)
		R17_Data: udt_Generic_Robot_20161202;				(*Global Data Area for R17 Input*)
		R18_Data: udt_Generic_Robot_20161202;				(*Global Data Area for R18 Input*)
		R19_Data: udt_Generic_Robot_20161202;				(*Global Data Area for R19 Input*)
		R20_Data: udt_Generic_Robot_20161202;				(*Global Data Area for R20 Input*)
		R21_Data: udt_Generic_Robot_20161202;				(*Global Data Area for R21 Input*)
		R22_Data: udt_Generic_Robot_20161202;				(*Global Data Area for R22 Input*)
		R23_Data: udt_Generic_Robot_20161202;				(*Global Data Area for R23 Input*)
		R24_Data: udt_Generic_Robot_20161202;				(*Global Data Area for R24 Input*)
		R25_Data: udt_Generic_Robot_20161202;				(*Global Data Area for R25 Input*)
		R26_Data: udt_Generic_Robot_20161202;				(*Global Data Area for R26 Input*)
		R27_Data: udt_Generic_Robot_20161202;				(*Global Data Area for R27 Input*)
		R28_Data: udt_Generic_Robot_20161202;				(*Global Data Area for R28 Input*)
		R29_Data: udt_Generic_Robot_20161202;				(*Global Data Area for R29 Input*)
		R30_Data: udt_Generic_Robot_20161202;				(*Global Data Area for R30 Input*)

	
		(* Data Frame Work for Interface to UI(s), be sure to see "Work Space" in Resources Tab for entitiy export*)
		(*Interfacing to all UI(s)*)
                 	In_From_ICxx: udt_UIcommon_Input_20250616;                    			(* Data Frame Work for Receiving Data from any IC -> NOTE:, also see Global_Persistent_Variables area*)
                 	Out_To_ICxx: udt_UIcommon_Output_20251008;                          	(* Data Frame Work for Sending Data to any IC*)


		EL6900_Connection_STAT AT %I*: ST_FSoE_14Byte;		(*Instance of Data Type Created so System Manager Can Use Type*)
		EL6692_In_Template AT %I*: udt_GenericRobot_AnyFieldbus_Input58Bytes;
		EL6692_Out_Template AT %Q*: udt_GenericRobot_AnyFieldbus_Output58Bytes;


END_VAR

// ---- Global Variables/Variable_Configuration.TcGVL
{attribute 'Tc2GvlVarNames'}
VAR_CONFIG
END_VAR

// ---- POUs/MAIN.TcPOU
(*!!!!!!!!!!!!!!!!!!!!!!!!!!!!!!!!!!!!!!!!!!!!!!!!!!!!!!!!!!!!!!!!!!!!!!!!!!!!!!!!!!!!!!!!!!!!!!!!!!!!!!!!!!!!!!!!!!!!!!!!!!!!!!!!!!!!!!!!!!!!!!!!!!!!!!!!!!!!
	Original Code Concept By: B.Lekx-Toniolo of Toniolo Research & Development Inc. 
	all copyright, IP and moral rights apply
	Date: July 2010.
	Fort Wisers
	S.H.H.D.I. 
	
	Major Migration from TC2 -> TC3 Platform primarily handled by Chris Drees of Sodecia GTAC 
	Date: 2020
	Major Migration from IWS -> TcHmi Platform primarily handled by c.drees and b.lekx-toniolo
	Date: 2022 - 2024
	
	
----------------------------------------------------------------------------------------------------------------------
REVISION NOTES: 
	Date: May 2012
	- generic functionality mods: Rob Remillard
	Date: December 2012
	- Various Updates to accomodate hardware change to SSCCv4.6 and allow Kuka and Motoman use, b.lekx-toniolo
	Date: May/June 2013
	- B562 As Commisioned for AB Ring, b.lekx-toniolo and r.remillard
	Date: July 2014
	- added robot capability of up to 20 robots, JVD
	- changed to allow up to 8 ICs wherever it was missing, JVD
	Date: October 2014
	- added capability of up to 30 robots maximum (25 recommended), b.lekx-toniolo
	Date: Summer / Fall 2015
	- migration to V5.00 machines (Win7 Platform), b.lekx-toniolo
	Date: Spring 2017
	- migration to V5.03 machines (Minor changes), b.lekx-toniolo
	Date: April 2017
	- Update to Kuka FB for new Safe Space, r.remillard
	Date: Summer/Fall 2017
	- migration to v5.04 machines (Minor changes), j.vandongen
	Date: Fall 2019
	- migration to v5.05 machines (Minor changes), j.vandongen
	- revamped the EOAT section, j.vandongen
	- changed ST from Nelson to Emhart. Nelson instance stored in the FB, j.vandongen
	Date: Fall/Winter 2019-2020
	- migration to v5.06 level as follows (also see task list for details)
		>production code updates per R&D request, b.lekx-toniolo, r.remillard, c.drees
		>brought in latest servo code, b.lekx-toniolo
		>various small bug fixes as per bug fix list, b.lekx-toniolo
		>Emhart code / UI upgrades (developed by j.underhill, imported by blt)
		>EOAT code / UI upgrades (developed by j.vandongen, imported by blt)
	Date: Winter 2020-2021
	- major migration from TC2 -> TC3 platform to create V6.xx level(c.drees, b.lekx-toniolo)
		>overhaul of safety from old config type to new visual layout (c.drees)
		>minor and various updates as required by new platform (c.drees, b.lekx-toniolo)
	Date: May 2021
	-Relinked all I/O link waterstands (c.drees)
	-corrected KUKA_FB version to ensure functionality is not missing (c.drees)
	-Corrected WS_FB version to ensure that functionality is not lost (c.drees)
	-Added All WCU Stepper reset checks and Any_TipChange_Request (c.drees)
	
	Date: 2022, 2023, 2024
	- IWS to TcHMI (TcUI) migration project, creates new rev level 6.10
		> various PLC changes as a result of migration work (b.lekx-toniolo / c.drees)
		> some PLC bug fixes while co-maintaining project PLC copy and SSCC6.01 (working FW package at time) (b.lekx-toniolo / c.drees)
	   	> Added Swing Arm control FBs to Main
		> added in various chages for project 90034 (simulation integration) (b.lekx-toniolo)

	
-----------------------------------------------------------------------------------------------------------------------
Some Key Notes Common to Project:
	All FBs and FUNs are 100% generic and thus exportable to other IC's of same version level (5.xx) (6.xx)
	All Prgs are custom per IPC (should not be exported)
------------------------------------------------------------------------------------------------------------------------
Some Notes for general mapping from Process Flow Department:
Fix#1-99 = Fixtures with Human Interaction
Fix#101-199 = Fixtures with NO Human Interaction (internal)
etc etc

------------------------------------------------------------------------------------------------------------------------
Some notes on Commenting Conventions
	Please everyone try to comment where you make changes / additions
	Some comment formats should be used where applicable / possible

	EXAMPLES:
		(*DEBUG, blah blah blah, your initials*)
			- this type of comment should be used where you've left something in a state that the end application deployment programmer needs to confirm/check/modify etc
				once they have done what they need to do, the comment should be deleted unless it's still applicable. The machine should be as free of DE BUG type comments before
				it ships to the end customer.

		(*NOTE, bling bling bling, your initials*)
			- this type of comment should be used when a specifc area of code might be of interest or value to the next anticipated person
				for example, if you've finished off some code as far as you can but know the next user will likely build upon it, a comment like this can be used.
				you may even co-ordinate with the end user and put their name or a keyword in place so they can search specific notes left for them
				this comment should not be used if the code is left in an unfinsihed state that may cause the machine to not run, in that case a DE BUG note shall be used

thanks to j.underhill for this comment convention contribution
------------------------------------------------------------------------------------------------------------------------
*)

PROGRAM MAIN
VAR

(*Establish Data Area for Mother Board Status Information*)
		Mother_Board AT%I*: udt_SMB_Status_20141211;
(*Establish FB for EtherCAT*)
		ECAT_Master: FB_GTAC_EtherCATMaster_20250723;

(*Establish Data Area for Ethernet Port*)
		DevState AT%I*:UINT;
(*Establish Data Area for System Time*)
		Get_LocalMachine_TimeFB: NT_GetTime;
		Local_Time: Timestruct;
(*Command to write all persistent data to the hard disk*)
		WritePersistent: WritePersistentData;
		DebugTime :TIME;
	
(*!!!!!!!!!!!!!!!!!!!!!!!!!!!!!!!!!!!!!!!!!!!!!!!!!!!!!!!!!!!!!!!!!!!!!!!!!!!!!!!! STOCK Variables - !!!DO NOT MODIFY !!!!!!!!!!!!!!!!!!!!!!!!!!!!!!!!!!!!!!!!!!!!!!!!!!!!!!!*)
		(*Main Scoped Variables*)
		Stay_Off: BOOL:= FALSE;
		Starting_Scan_PulseTMR: TON;
		Starting_Scan_Pulse: BOOL;	(*1.0ms Pulse that Occurs at Boot-Up*)

		All_Estops_OK AT %I*: BOOL;
		All_SafetyGates_OK AT %I*: BOOL;
		Control_Power_ON: BOOL;
		All_EStopRLYs_Off: BOOL;
		SAFETY_RESET: BOOL;
		All_RobotsReady_Running: BOOL;

		Safety_Zone_Test AT %Q*: BOOL;
		Roll_Door01_Enable AT %I*: BOOL;
		Roll_Door02_Enable AT %I*: BOOL;
		Access_Violation AT %I*: BOOL;
		
		(*ADDED TO RETRIEVE DATA FROM ALL IC's - AB*)
		Access_Violation_IC01 AT %I*: BOOL;
		Access_Violation_IC02 AT %I*: BOOL;
		Access_Violation_IC03 AT %I*: BOOL;
		
		(*Verti Guard IO*)
		VertiGuard_N01 AT %Q*: udt_EP2028_002_v2;
		VertiGuard_N01_STAT AT %I*: udt_EP2028_002_STAT;
		VertiGuard_N02 AT %I*: udt_EP1908_002;

		(*Prog OK Status Bits*)
		Safety_Reset_ProgOK: BOOL;
		Robot_Interf_Map_ProgOK: BOOL;
		TipChange_ProgOK: BOOL;
		Faults_ProgOK: BOOL;
		UI_ProgOK: BOOL;
		
		(*Hardware Diagnostic Data*)
		HardwareStat:FB_SystemDiags20241206;
		ApplicationData:PlcAppSystemInfo;
		Taskdata:PLCTaskSystemInfo;
		
		(*TLK ADDED FOR MD DOORS CLOSE FEEDBACK*)
		MD01_N01_I0 AT %I*: BOOL;
		MD01_N01_I1 AT %I*: BOOL;
		MD01_N01_I2 AT %I*: BOOL;
		MD01_N01_I3 AT %I*: BOOL;
		
		MD02_N01_I0 AT %I*: BOOL;
		MD02_N01_I1 AT %I*: BOOL;
		MD02_N01_I2 AT %I*: BOOL;
		MD02_N01_I3 AT %I*: BOOL;
		
		
(*$$$$$$$$$$$$$$$$$$$$$$ NON Stock Variables, Instances etc (add here as you add robots and fixtures) $$$$$$$$$$$$$$$$$$$$$$$$$$$$$$$$$$$$$$*)
		(*IS Instances*)
		IS01: FB_GTAC_ISxx_20241121;			(*IS01*)

		(*IC Instances*)
		IC01: FB_GTAC_ICxx_20181023;				(*IC01*)
		IC02: FB_GTAC_ICxx_20181023;				(*IC02*)
		IC03: FB_GTAC_ICxx_20181023;				(*IC03*)
		IC04: FB_GTAC_ICxx_20181023;				(*IC04*)
		IC05: FB_GTAC_ICxx_20181023;				(*IC05*)
		IC06: FB_GTAC_ICxx_20181023;				(*IC06*)
		IC07: FB_GTAC_ICxx_20181023;				(*IC07*)
		IC08: FB_GTAC_ICxx_20181023;				(*IC08*)

		(*Robot Instances*)
		(*R1: FB_GTAC_Motoman_20151105;	*)		(*EXAMPLE!!! Robot is MOTO DX100 32 Byte Type*)
		R1: FB_GTAC_Kuka_CUSTOM;		(*Robot is KUKA KRC4 Type*)
		R2: FB_GTAC_Kuka_CUSTOM;		(*Robot is KUKA KRC4 Type*)
		R3: FB_GTAC_Kuka_CUSTOM;		(*Robot is KUKA KRC4 Type*)
		R4: FB_GTAC_Kuka_CUSTOM;		(*Robot is KUKA KRC4 Type*)
		R5: FB_GTAC_Kuka_CUSTOM;		(*Robot is KUKA KRC4 Type*)
		R6: FB_GTAC_Kuka_CUSTOM;		(*Robot is KUKA KRC4 Type*)
		R7: FB_GTAC_Kuka_CUSTOM;		(*Robot is KUKA KRC4 Type*)
		R8: FB_GTAC_Kuka_CUSTOM;		(*Robot is KUKA KRC4 Type*)
		R9: FB_GTAC_Kuka_CUSTOM;		(*Robot is KUKA KRC4 Type*)
		R10: FB_GTAC_Kuka_CUSTOM;		(*Robot is KUKA KRC4 Type*)
		R11: FB_GTAC_Kuka_CUSTOM;		(*Robot is KUKA KRC4 Type*)
		R12: FB_GTAC_Kuka_CUSTOM;		(*Robot is KUKA KRC4 Type*)
		R13: FB_GTAC_Kuka_CUSTOM;		(*Robot is KUKA KRC4 Type*)
		R14: FB_GTAC_Kuka_CUSTOM;		(*Robot is KUKA KRC4 Type*)
		R15: FB_GTAC_Kuka_CUSTOM;		(*Robot is KUKA KRC4 Type*)
		R16: FB_GTAC_Kuka_CUSTOM;		(*Robot is KUKA KRC4 Type*)
		R17: FB_GTAC_Kuka_CUSTOM;		(*Robot is KUKA KRC4 Type*)
		R18: FB_GTAC_Kuka_CUSTOM;		(*Robot is KUKA KRC4 Type*)
		R19: FB_GTAC_Kuka_CUSTOM;		(*Robot is KUKA KRC4 Type*)
		R20: FB_GTAC_Kuka_CUSTOM;		(*Robot is KUKA KRC4 Type*)
		R21: FB_GTAC_Kuka_CUSTOM;		(*Robot is KUKA KRC4 Type*)
		R22: FB_GTAC_Kuka_CUSTOM;		(*Robot is KUKA KRC4 Type*)
		R23: FB_GTAC_Kuka_CUSTOM;		(*Robot is KUKA KRC4 Type*)
		R24: FB_GTAC_Kuka_CUSTOM;		(*Robot is KUKA KRC4 Type*)
		R25: FB_GTAC_Kuka_CUSTOM;		(*Robot is KUKA KRC4 Type*)
		R26: FB_GTAC_Kuka_CUSTOM;		(*Robot is KUKA KRC4 Type*)
		R27: FB_GTAC_Kuka_CUSTOM;		(*Robot is KUKA KRC4 Type*)
		R28: FB_GTAC_Kuka_CUSTOM;		(*Robot is KUKA KRC4 Type*)
		R29: FB_GTAC_Kuka_CUSTOM;		(*Robot is KUKA KRC4 Type*)
		R30: FB_GTAC_Kuka_CUSTOM;		(*Robot is KUKA KRC4 Type*)

		
		
		
		SS01: FB_GTAC_SS_20250407;										(*Large Type Services Stand*)
		SS02: FB_GTAC_SS_20250407;										(*Large Type Services Stand*)
		SS03: FB_GTAC_SS_20250407;										(*Large Type Services Stand*)

		ESW01: FB_GTAC_ESW_20150814;									(*Enabling Switch Option Plate*)
		ESW02: FB_GTAC_ESW_20150814;									(*Enabling Switch Option Plate*)
		ESW03: FB_GTAC_ESW_20150814;									(*Enabling Switch Option Plate*)
		ESW04: FB_GTAC_ESW_20150814;									(*Enabling Switch Option Plate*)

		ST01: FB_Emhart_20200113;										(*Stud Contoller*)
		ST02: FB_Emhart_20200113;										(*Stud Contoller*)
		ST03: FB_Emhart_20200113;										(*Stud Contoller*)
		ST04: FB_Emhart_20200113;										(*Stud Contoller*)
		ST05: FB_Emhart_20200113;										(*Stud Contoller*)

		SL01: FB_Graco_Seal_20200716;								(*Sealant Controller*)
		SL02: FB_Graco_Seal_20200716;								(*Sealant Controller*)
		SL03: FB_Graco_Seal_20200716;								(*Sealant Controller*)
		SL04: FB_Graco_Seal_20200716;								(*Sealant Controller*)

		NutWeld_LVDT: ARRAY [0..5] OF FB_GTAC_NutWeldLVDT_20250612;		(*Nut Weld Based LVDT Systems*)
		
				SIC01: FB_SIC_MarkProfi_20200727;
		SIC02: FB_SIC_MarkProfi_20200727;

		Laser01: FB_Trumpf_20180125;								(*Laser Controller*)

		RollDoor01: FB_GTAC_RollDoor_20190108;						(*Roll Up Door - Old Style*)
		MD01: FB_GTAC_MDxx_20251008;								(*Motorized Roll Up Door - New Style*)
		MD02: FB_GTAC_MDxx_20251008;								(*Motorized Roll Up Door - New Style*)
		MD03: FB_GTAC_MDxx_20251008;								(*Motorized Roll Up Door - New Style*)
		MD04: FB_GTAC_MDxx_20251008;								(*Motorized Roll Up Door - New Style*)
		MD05: FB_GTAC_MDxx_20251008;								(*Motorized Roll Up Door - New Style*)

		Conveyor01: FB_GTAC_Conveyor_20210303;						(*Conveyor*)
		VFD01: FB_SCHNEIDERVFD_20180808;							(*Stand alone VFD*)
		VFD02: FB_SCHNEIDERVFD_20180808;							(*Stand alone VFD*)
		VFD03: FB_SCHNEIDERVFD_20180808;							(*Stand alone VFD*)
		VFD04: FB_SCHNEIDERVFD_20180808;							(*Stand alone VFD*)
		VFD05: FB_SCHNEIDERVFD_20180808;							(*Stand alone VFD*)
		
		(*FB Ok Status Bits*)
		IC01_FBOK: BOOL;
		IC02_FBOK: BOOL;
		IC03_FBOK: BOOL;
		IC04_FBOK: BOOL;
		IC05_FBOK: BOOL;
		IC06_FBOK: BOOL;
		IC07_FBOK: BOOL;
		IC08_FBOK: BOOL;

		R1_FBOK: BOOL;
		R2_FBOK: BOOL;
		R3_FBOK: BOOL;
		R4_FBOK: BOOL;
		R5_FBOK: BOOL;
		R6_FBOK: BOOL;
		R7_FBOK: BOOL;
		R8_FBOK: BOOL;
		R9_FBOK: BOOL;
		R10_FBOK: BOOL;
		R11_FBOK: BOOL;
		R12_FBOK: BOOL;
		R13_FBOK: BOOL;
		R14_FBOK: BOOL;
		R15_FBOK: BOOL;
		R16_FBOK: BOOL;
		R17_FBOK: BOOL;
		R18_FBOK: BOOL;
		R19_FBOK: BOOL;
		R20_FBOK: BOOL;
		R21_FBOK: BOOL;
		R22_FBOK: BOOL;
		R23_FBOK: BOOL;
		R24_FBOK: BOOL;
		R25_FBOK: BOOL;
		R26_FBOK: BOOL;
		R27_FBOK: BOOL;
		R28_FBOK: BOOL;
		R29_FBOK: BOOL;
		R30_FBOK: BOOL;

		(*Ped Stations*)
		Ped: ARRAY [0..30] OF  FB_GTAC_Ped_20240808;
 	
		(*Rising Edge Triggers*)
		RPulse: ARRAY [0..31] OF  R_TRIG;
	
	
	(*temp debug bits*)
	debug_test1: BOOL;
	debug_test2: BOOL;
	
	TEST1: BOOL;
	test2: UINT;
	
	VertiGuard_1: FB_VertiGuard_20260310;
	
	
END_VAR


(*VAR_INPUT
	(*OPC / Simulation Vars*)
	{attribute 'OPC.UA.DA':='1'}
	SIM_WorkAround_StartRobots: BOOL;
	{attribute 'OPC.UA.DA':='1'}
	SIM_WorkAround_StartFix01: BOOL;
	{attribute 'OPC.UA.DA':='1'}
	SIM_WorkAround_StartFix02: BOOL;
	{attribute 'OPC.UA.DA':='1'}
	SIM_WorkAround_StartFix03: BOOL;
	{attribute 'OPC.UA.DA':='1'}
	SIM_WorkAround_StartFix04: BOOL;
	{attribute 'OPC.UA.DA':='1'}
	SIM_WorkAround_StartFix05: BOOL;
	{attribute 'OPC.UA.DA':='1'}
	SIM_WorkAround_StartFix06: BOOL;
	{attribute 'OPC.UA.DA':='1'}
	SIM_WorkAround_StartFix07: BOOL;
	{attribute 'OPC.UA.DA':='1'}
	SIM_WorkAround_StartFix08: BOOL;
	{attribute 'OPC.UA.DA':='1'}
	SIM_WorkAround_StartFix09: BOOL;
	{attribute 'OPC.UA.DA':='1'}
	SIM_WorkAround_StartFix10: BOOL;
	{attribute 'OPC.UA.DA':='1'}
	SIM_WorkAround_StartFix11: BOOL;
	{attribute 'OPC.UA.DA':='1'}
	SIM_WorkAround_StartFix12: BOOL;
	{attribute 'OPC.UA.DA':='1'}
	SIM_WorkAround_StartFix13: BOOL;
	{attribute 'OPC.UA.DA':='1'}
	SIM_WorkAround_StartFix14: BOOL;
	{attribute 'OPC.UA.DA':='1'}
	SIM_WorkAround_StartFix15: BOOL;
	{attribute 'OPC.UA.DA':='1'}
	SIM_WorkAround_StartFix16: BOOL;

	{attribute 'OPC.UA.DA':='1'}
	SIM_WorkAround_StartFix101: BOOL;
	{attribute 'OPC.UA.DA':='1'}
	SIM_WorkAround_StartFix102: BOOL;
	{attribute 'OPC.UA.DA':='1'}
	SIM_WorkAround_StartFix103: BOOL;
	{attribute 'OPC.UA.DA':='1'}
	SIM_WorkAround_StartFix104: BOOL;
	{attribute 'OPC.UA.DA':='1'}
	SIM_WorkAround_StartFix105: BOOL;
	{attribute 'OPC.UA.DA':='1'}
	SIM_WorkAround_StartFix106: BOOL;
	{attribute 'OPC.UA.DA':='1'}
	SIM_WorkAround_StartFix107: BOOL;
	{attribute 'OPC.UA.DA':='1'}
	SIM_WorkAround_StartFix108: BOOL;
	{attribute 'OPC.UA.DA':='1'}
	SIM_WorkAround_StartFix109: BOOL;
	{attribute 'OPC.UA.DA':='1'}
	SIM_WorkAround_StartFix110: BOOL;
	{attribute 'OPC.UA.DA':='1'}
	SIM_WorkAround_StartFix111: BOOL;
	{attribute 'OPC.UA.DA':='1'}
	SIM_WorkAround_StartFix112: BOOL;

	{attribute 'OPC.UA.DA':='1'}
	SIM_WorkAround_GeneralInputs: ARRAY[0..31] OF BOOL;
	
	{attribute 'OPC.UA.DA':='1'}
	SIM_WorkAround_TT01_Position_Index: ARRAY[0..1] OF BOOL;
	{attribute 'OPC.UA.DA':='1'}
	SIM_WorkAround_TT02_Position_Index: ARRAY[0..1] OF BOOL;
	{attribute 'OPC.UA.DA':='1'}
	SIM_WorkAround_TT03_Position_Index: ARRAY[0..1] OF BOOL;
	{attribute 'OPC.UA.DA':='1'}
	SIM_WorkAround_TT04_Position_Index: ARRAY[0..1] OF BOOL;
	{attribute 'OPC.UA.DA':='1'}
	SIM_WorkAround_TT05_Position_Index: ARRAY[0..1] OF BOOL;
	{attribute 'OPC.UA.DA':='1'}
	SIM_WorkAround_TT06_Position_Index: ARRAY[0..1] OF BOOL;
	{attribute 'OPC.UA.DA':='1'}
	SIM_WorkAround_TT07_Position_Index: ARRAY[0..1] OF BOOL;
	{attribute 'OPC.UA.DA':='1'}
	SIM_WorkAround_TT08_Position_Index: ARRAY[0..1] OF BOOL;
	{attribute 'OPC.UA.DA':='1'}
	SIM_WorkAround_TT09_Position_Index: ARRAY[0..1] OF BOOL;
	{attribute 'OPC.UA.DA':='1'}
	SIM_WorkAround_TT10_Position_Index: ARRAY[0..1] OF BOOL;
	{attribute 'OPC.UA.DA':='1'}
	SIM_WorkAround_FixXx_LoadParts: ARRAY[0..112] OF ARRAY[0..15] OF BOOL;
	{attribute 'OPC.UA.DA':='1'}
	SIM_WorkAround_FixXx_OpPower: ARRAY[0..112] OF BOOL;
	{attribute 'OPC.UA.DA':='1'}
	SIM_WorkAround_FixNumberAndModel: ARRAY[1..112] OF ARRAY[0..15] OF BOOL;
	(*Used for setting model in above array - See SIM Action under GTAC_CONFIG*)
	i: INT;
	j: INT;
	Fix01PrevModelId: INT:= 0; 
	Fix02PrevModelId: INT:= 0; 
	Fix03PrevModelId: INT:= 0; 
	Fix04PrevModelId: INT:= 0; 
	{attribute 'OPC.UA.DA':='1'}
	SIM_WorkAround_FixXx_HandClamp: ARRAY[0..112] OF BOOL;

	(*Added Custom for this machine for R04 Linear Rail animation, blt (Will's code*)
	SIM_ExternalAxis_Control: INT;

END_VAR*)

(*Develop 5.0ms Pulse for Reseting System During Boot-Up*)
	Starting_Scan_PulseTMR.PT:= T#5MS;
	Starting_Scan_PulseTMR.IN:= TRUE;
	Starting_Scan_PulseTMR();
	Starting_Scan_Pulse:= NOT Starting_Scan_PulseTMR.Q;

(*Send Mother Board Status, Task Data and Application Data to UI*)
	Out_To_ICxx.Appdata:= _AppInfo;
	Out_To_ICxx.TaskData:= _TaskInfo[1];
	
	(*Call TC3 required HW diag FB (not previouslly required in TC2)*)
	HardwareStat();
	Out_To_ICxx.MboardData:= HardwareStat.HardwareDiag;		

	
(*EtherCAT Master*)
	(*Inputs*)
	ECAT_Master.Blank_Config_Trigger:= Starting_Scan_Pulse;	 																(*Upon first start, blank config array*)
	ECAT_Master.Read_Config_Trigger:= NOT Starting_Scan_Pulse AND Pulse_CoERead AND NOT Out_To_ICxx.ControlPower1_OK;		(*When machine is past first scan, read config (except if runnng)*)
	ECAT_Master.Read_States_Trigger:= NOT Starting_Scan_Pulse AND Pulse_1S;
	ECAT_Master.Machine_Running:= Out_To_ICxx.ControlPower1_OK;									(*Stop Config Reads when Machne is ready to run*)
		(*Overrides may be placed immediatly after components automatically found in EtherCAT configuration
		the overrides are used to force display of Components created manually in the UIs but are not part of the standard set
		of components coded in the EtherCAT Master FB*)
		ECAT_Master.ComponentConfig_Overrides[41]:='SL01';
		ECAT_Master.ComponentConfig_Overrides[42]:='SL02';
		ECAT_Master.ComponentConfig_Overrides[43]:='SL03';
		ECAT_Master.ComponentConfig_Overrides[44]:='SL04';
		ECAT_Master.ComponentConfig_Overrides[45]:='LSR01';		
		ECAT_Master.ComponentConfig_Overrides[46]:='LSR02';		
	(*Actual Call*)
	ECAT_Master();
	(*Outputs*)
	(*Send Ecat Master Status to UIs*)
	Out_To_ICxx.EtherCat_Master_Image:= ECAT_Master.Discrete_Image;



(*$$$$$$$$$$$$$$$$$$$$$$$$$$$$$$$$$$$$$$$$$$$$$$$$$$ The Main Progam $$$$$$$$$$$$$$$$$$$$$$$$$$$$$$$$$$$$$$$$$$$$$$$$$$$$*)
(*--------------------------------------------------------------------------------------- GTAC CONFIG -----------------------------------------------------------------------------------------------*)
	(*Run the Config to retreive Data for Code Re-action*)
	GTAC_CONFIG();

		Out_To_ICxx.Machine_Serial:= GTAC_CONFIG.Machine_Serial;
		Out_To_ICxx.Machine_Common_Name:= GTAC_CONFIG.Machine_Common_Name;
		Out_To_ICxx.Machine_Build_Used:= GTAC_Config.Machine_Build_Used;
		Out_To_ICxx.Machine_Appl_Dev:= GTAC_Config.Machine_Appl_Dev;
		(*Production Related Configuration Data to UI*)
		Out_To_ICxx.ProdConfig_Target_CycleTime:= GTAC_CONFIG.ProdConfig_Target_CycleTime;
		Out_To_ICxx.ProdConfig_Common:= GTAC_CONFIG.ProdConfig_Common;
		Out_To_ICxx.ProdConfig_Day:= FUN_GTAC_TODtoUDINT(GTAC_CONFIG.ProdConfig_Day);
		Out_To_ICxx.ProdConfig_Aft:= FUN_GTAC_TODtoUDINT(GTAC_CONFIG.ProdConfig_Aft);
		Out_To_ICxx.ProdConfig_Mid:= FUN_GTAC_TODtoUDINT(GTAC_CONFIG.ProdConfig_Mid);
		(*Machine Related Configuration Data to UI*)
		Out_To_ICxx.Option_Air1:= GTAC_CONFIG.Option_Air1;
		Out_To_ICxx.Option_Air2:= GTAC_CONFIG.Option_Air2;
		Out_To_ICxx.Option_Water1:= GTAC_CONFIG.Option_Water1;
		Out_To_ICxx.Option_Water2:= GTAC_CONFIG.Option_Water2;
		Out_To_ICxx.Option_WaterTimeOut_Enable:= GTAC_CONFIG.Option_WaterTimeOut_Enable;
		Out_To_ICxx.Option_WaterFlowTimeOut_SP:= GTAC_CONFIG.Option_WaterFlowTimeOut_SP;
		Out_To_ICxx.Option_WaterTempHighLimit1:= GTAC_CONFIG.Option_WaterTempHighLimit1;
		Out_To_ICxx.Option_WaterTempHighLimit2:= GTAC_CONFIG.Option_WaterTempHighLimit2;
		Out_To_ICxx.Option_WaterFlowLowLimit1:= GTAC_CONFIG.Option_WaterFlowLowLimit1;
		Out_To_ICxx.Option_WaterFlowLowLimit2:= GTAC_CONFIG.Option_WaterFlowLowLimit2;
		Out_To_ICxx.Option_ESW_Count:= GTAC_CONFIG.Option_ESW_Count;
		Out_To_ICxx.Option_MD_Count:= GTAC_CONFIG.Option_MD_Count;
		Out_To_ICxx.Option_IS_Count:= GTAC_CONFIG.Option_IS_Count;
		Out_To_ICxx.Option_IC_Count:= GTAC_CONFIG.Option_IC_Count;
		Out_To_ICxx.Option_HumanFix_Enables:= GTAC_CONFIG.Option_HumanFix_Enables;
		Out_To_ICxx.Option_InternalFix_Count:= GTAC_CONFIG.Option_InternalFix_Count;
		Out_To_ICxx.Option_Robot_Count:= GTAC_CONFIG.Option_Robot_Count;
		Out_To_ICxx.Option_Ped_Count:= GTAC_CONFIG.Option_Ped_Count;
		Out_To_ICxx.Option_SealController_Count:= GTAC_CONFIG.Option_SealController_Count;
		Out_To_ICxx.Option_StudController_Count:= GTAC_CONFIG.Option_StudController_Count;
		Out_To_ICxx.Option_NutWelder_Count:= GTAC_CONFIG.Option_NutWelder_Count;
		Out_To_ICxx.Option_SD_Count:= GTAC_CONFIG.Option_SD_Count;
		Out_To_ICxx.Option_VFD_Count:= GTAC_CONFIG.Option_VFD_Count;
		Out_To_ICxx.Config_Fault:= GTAC_CONFIG.Fault;

		(*Various Development States to UI*)
		Out_To_ICxx.InDryCycle:= GTAC_CONFIG.Dry_Cycle_Enabled;
		IF NOT GTAC_CONFIG.Dry_Cycle_Enabled
			THEN
			Out_To_ICxx.In_Local_DryCycle:= GTAC_CONFIG.Local_DryCycle_Enables;
		ELSIF GTAC_CONFIG.Dry_Cycle_Enabled
			THEN
			Out_To_ICxx.In_Local_DryCycle:= 131070;		(*Set Bits .1 through .16 high to annunciate dry cycle on those tools*)
		END_IF;

		Out_To_ICxx.In_Low_Speed:=GTAC_CONFIG.Low_Speed_Enabled;
		Out_To_ICxx.Under_Construction:= GTAC_CONFIG.Under_Construction;
		Out_To_ICxx.In_Sim_Mode:= GTAC_CONFIG.In_SIM_Mode;
		Out_To_ICxx.CycleHold_OK:=  In_From_ICxx.Cycle_Hold;

		(*This Overrides the T1 zone disable so robot programmers can verify the monitoring space dimensions*)
		Safety_Zone_Test:= In_From_ICxx.T1_Zone_Test;
		Out_To_ICxx.T1_Zone_Test_ACK:= Safety_Zone_Test;

(*----------------------------------------------------------------------------- Main Status Of Machine Control Power-------------------------------------------------------------------------*)
	(*Estops*)
	Out_To_ICxx.Estops_OK:= All_Estops_OK; (*All_Estops_OK is a linked var in System Manager and is to be linked to Output of TwinSAFE FB in IC01 Called "Gather All Estops" (FB20)*)

	(*!!!All_EstopRLYs_Off is left to configure at Application Deployment time and not auto configured by GTAC Options!!!*)
	All_EstopRLYs_Off:=
						IS01.Estop_Relays_Off AND
						SS01.Valves_Off AND
						R1.Estop_Relays_Off AND R2.Estop_Relays_Off AND
						R3.Estop_Relays_Off AND R4.Estop_Relays_Off AND
						R5.Estop_Relays_Off AND R6.Estop_Relays_Off AND
						R7.Estop_Relays_Off AND R8.Estop_Relays_Off AND
						R9.Estop_Relays_Off AND R10.Estop_Relays_Off AND
						R11.Estop_Relays_Off;


	(*Safety Gates*)
	IC01.FB_In.Output_Req1:= In_From_ICxx.LockSGK1;
	Out_To_ICxx.Safety_Gates_OK:= All_SafetyGates_OK; (*All_SafetyGates_OK is a linked var in System Manager and is to be linked to Output of TwinSAFE FB in IC01 Called "Gather All Gates (FB35)*)

	(*OverAll Control Power Status*)
	Control_Power_ON:= All_Estops_Ok AND All_SafetyGates_OK AND
						((IS01.Estop_Relays_On AND IS01.Gate_Relays_On) OR GTAC_CONFIG.Option_IS_Count<1);

	Out_To_ICxx.ControlPower1_OK:= Control_Power_ON;

(*------------------------------------------------------------------------ Develop Safety Reset ---------------------------------------------------------------------------------------------------*)

	IF All_Estops_OK
		THEN
			SAFETY_RESET:= In_From_ICxx.ControlPower1;
	ELSIF NOT All_Estops_Ok AND All_EstopRLYs_Off
		THEN
			SAFETY_RESET:= In_From_ICxx.ControlPower1;                               (*Ensure no Estop Relays Are Stuck In On Position*)
	END_IF (*NOTE*)

(*!!!!!!!!!! use this to do the first reset !!!!!!!!!!!!!!!!!!*)
	SAFETY_RESET;

(*
NOTE - You should note that this is the one and only location that the semi colon is NOT used to close a conditional block of code.
That should lead you to note that the TCAT compiler will accept both cases (with and without semi colon closure).
So, which is more correct? There are two frames of thought:
	1. The semi is used to close every other piece of code outside of conditional statement blocks, therefore, for consistency, the semi is correct.
		Also, most documents pertaining to ST show the semi in place, offering more validity to the consistency argument.
		The semi was also required in legacy compilers such as Turbo Pascal, so the semi at the end of conditional code blocks also has historical value. 
	2. Syntactically, the semi is not required by the compiler. A semi found in this position by the compiler results in no actual CPU instruction generation so it's simply
		one more line the compiler must scan and "throw away".  So if we don't want to use it from a syntax perspective, then we should not be using it on any closure of a conditional
		block of code for consistency sake. However, please keep in mind that a semi not found in other places will be considered an error.
		So, if consistency is to be our driving force then, from a global syntax point of view, a semi is more valid as all other lines of code require semi closure (IE digression to point 1).
		So the only reason left is to avoid extra compiler load, which does hold some value. 
		However, I timed the compiler both with and without the semi and found no real difference (accurate to maybe +- 1  sec).

In this case both answers have some merit in "correctness". 
However I believe the argument clearly favors the points brought up in frame of thought 1.
The real value of this note is to spark an idea of digging deeper to find out the truth behind things and always ask "WHY".
Kudos to anyone who actually noticed the "semi colon paradox"
*)


	
(*------------------------------------------------------------------------- General Status Of Robots Within Machine -----------------------------------------------------------------------*)
	All_RobotsReady_Running:= (R1.Ready AND R1.Operating AND NOT R1.Faulted) AND
								(R2.Ready AND R2.Operating AND NOT R2.Faulted) AND
								(R3.Ready AND R3.Operating AND NOT R3.Faulted) AND
								(R4.Ready AND R4.Operating AND NOT R4.Faulted) AND
								(R5.Ready AND R5.Operating AND NOT R5.Faulted) AND
								(R6.Ready AND R6.Operating AND NOT R6.Faulted) AND
								(R7.Ready AND R7.Operating AND NOT R7.Faulted) AND
								(R8.Ready AND R8.Operating AND NOT R8.Faulted) AND
								(R9.Ready AND R9.Operating AND NOT R9.Faulted) AND
								(R10.Ready AND R10.Operating AND NOT R10.Faulted) AND
								(R11.Ready AND R11.Operating AND NOT R11.Faulted);


(*---------------------------------------------------------------------------------- Some General Purpose Code -------------------------------------------------------------------------------*)
	(*Pulse Generators*)
		(*1 Second On and Off Time*)
		Pulse_1S_FB.On_Time:=T#1.0S;
		Pulse_1S_FB.Off_Time:=T#1.0S;
		Pulse_1S_FB();
		Pulse_1S:=Pulse_1S_FB.Wave;
		(*0.5 Second On and Off Time*)
		Pulse_500ms_FB.On_Time:=T#500MS;
		Pulse_500ms_FB.Off_Time:=T#500MS;
		Pulse_500ms_FB();
		Pulse_500ms:=Pulse_500ms_FB.Wave;
		(*Pulse to Set Interval of CoE Reads*)
		Pulse_CoERead_FB.On_Time:=T#1S;
		Pulse_CoERead_FB.Off_Time:=T#30S;
		Pulse_CoERead_FB();
		Pulse_CoERead:=Pulse_CoERead_FB.Wave;

		(*Status Of PLC Running to UI (User Interface) "PLC Running" Indicator on all UI "IC01 Controls Overview" Screens*)
		Out_To_ICxx.Spare1:= TRUE;

(*--------------------------------------------------------------------------- Call Programs ---------------------------------------------------------------*)
(*Get Windows Time From Local Machine for Generating Production Report Frame Work*)
	Get_LocalMachine_TimeFB.START:= Pulse_500mS;
	Get_LocalMachine_TimeFB();
	Local_Time:= Get_LocalMachine_TimeFB.TIMESTR;

(*Call Fault Routine*)
	Faults();
	Out_To_ICxx.Faults_OK:= NOT Faults.System_Major_Fault; 					(*Pass Status to UI to drive Fault Warning Icon on General Status Object*)
	Out_To_ICxx.Overall_Controls_Fault.0:= Faults.General_Controls_Fault; 	(*Pass Status to UI to drive Red Flashing Prompt on Controls Icon*)
	
(*Call Robot InterLock_Map*)
	Robot_InterLock_Map();
(*Generate Task_ID Record*)
	Task_ID_Record();
(*Cell Services (Master Test, Brake Test, Tip Change, Tip Dress)*)
	(*Input Data*)
	Cell_Services_Prog.Enable_Motion:= All_Estops_OK;
	Cell_Services_Prog.Discrete_In.ModelData:= 1; (*Override to have single point selection*)
	Cell_Services_Prog.Discrete_In.ResetProd:= In_From_ICxx.Reset_ChangeCount;
	(*Call PROGRAM*)
	Cell_Services_Prog();
	(*Output Data*)
	Out_To_ICxx.MasterTest_Req_OK:= Cell_Services_Prog.Start_All_MTRobots;
	Out_To_ICxx.BrakeTest_Req_OK:= Cell_Services_Prog.Start_All_BTRobots;
	Out_To_ICxx.TipChangeReq_OK:= Cell_Services_Prog.Start_All_TCRobots;
	//Out_To_ICxx.Change_Count:= Cell_Services_Prog.Prod_Count_Out;
	Out_To_ICxx.Rxx_ReadyFor_TipChange:= Cell_Services_Prog.Rxx_ReadyAt_TipChangePosition;
Out_To_ICxx.Change_Count.2:= TRUE;
(* ------------------------------------------------------------------------------------- Ancillary Devices --------------------------------------------------------------------------------------------*)
(*Ped Stations*)
	Ped_Stations();

(*Ancillary Equipment such as Stud and Sealant Controllers*)
	Ancillary_Equipment();

(*Servo Motion Devices*)
IF GTAC_CONFIG.Option_SD_Count>0
	THEN
	Servo_Motion();
END_IF;

MAIN.VertiGuard_N01.Q.0:= MAIN.VertiGuard_1.GateClose_CMD;
MAIN.VertiGuard_N01.Q.1:= MAIN.VertiGuard_1.GateOpen_CMD;
(*-----------------------------------------------------------------------------------------------------------------------------------------------------------------------------------*)
(*----------------------------------------------------------------------- Invoke and Call Function Blocks -----------------------------------------------------------*)
(*-----------------------------------------------------------------------------------------------------------------------------------------------------------------------------------*)

(*----------------------------------------------------------------------------------------------------------------------------------------*)
(*Invoke IS FB*)
(*----------------------------------------------------------------------------------------------------------------------------------------*)
	(*IPC(IC) Supply Cabinet 01*)
	(*Input Data*)
	IS01.FB_In.Safety_RST:= SAFETY_RESET;
	IS01.FB_In.Enable_Motion:= All_Estops_OK AND All_SafetyGates_OK;
	IS01.FB_In.CoE_Read_Trigger:= (GTAC_CONFIG.Option_IC_Count>=1) AND Pulse_CoERead;	(*Global Interval of CoE Reads*)
	IS01.FB_In.Ecat_Master_AmsNetID:= MAIN.ECAT_Master.AmsID;
	IS01.FB_In.Prev_EcatNode_Present:= NOT ESW02.EP1908_NotPresent; 					(*Ensure Previous Node Exists to determine Ecat Cable Break of this Devices Input Cable*)
	IS01.FB_In.Option_Enable_SplitRelays:= TRUE;									(*Enable Split Relays Option, otherwise only power relays will be expected*)
	IS01.FB_In.Option_Enable_Pbus:= TRUE;											(*Enable EL6731 in PD if a profibus master is present. if not set to false*)
	(*Call FUNCTION*)
	IS01();
	(*Output Data*)
	Out_To_ICxx.IS[1].Discrete_Image:= IS01.Discrete_Image;
	Out_To_ICxx.IS[1].ECAT_Cable_Breaks:= IS01.EcatSlave_Cable_Breaks;
	
		

